(* IEC 61131-3 sources: MotionTestBenchMaster/Logical/00_AID/Libraries/Sidel_Libraries/Sidel (part 2) *)

(* ---- PID_FB.st ---- *)
FUNCTION_BLOCK PID_Cont
	VAR_RTInfo(enable:=TRUE);
	VAR_CycleCounter	:= MAX(1, VAR_CycleCounter + 1);

	TON_Cycle(	IN := TRUE,
				PT := IN_CycleTime - UDINT_TO_TIME(VAR_RTInfo.cycle_time / 1000));

	IF NOT TON_Cycle.Q THEN
		RETURN;
	END_IF

	VAR_CycleTime	:= (UDINT_TO_REAL(VAR_RTInfo.cycle_time) * VAR_CycleCounter) / 1000000.0;
	VAR_CycleCounter 	:= 0.0;
	memset(ADR(TON_Cycle), 0, SIZEOF(TON_Cycle));

	(*****************************************************************)
	(*************************SP MANAGE*******************************)
	(*****************************************************************)
	IF NOT VAR_FirstCycle THEN
		VAR_FirstCycle	:= TRUE;
		HMI.SPLocal		:= FALSE;
		OUT		:= 0.0;
		OUT_P	:= 0.0;
		OUT_I	:= 0.0;
		OUT_D	:= 0.0;
	END_IF

	IF EDGE(HMI.SPLocal) OR EDGEPOS(IN_Auto) THEN
		VAR_SlewInit	:= TRUE;
	END_IF

	IF VAR_SlewInit AND HMI.SPLocal THEN
		HMI.PV		:= IN_PV;
		LCRRamp.x	:= MIN(IN_PV, HMI.SP_Local);
		LCRRamp.set	:= TRUE;
	ELSIF VAR_SlewInit AND IN_Auto THEN
		HMI.PV		:= IN_PV;
		LCRRamp.x	:= MIN(IN_PV, IN_AutoSP);
		LCRRamp.set	:= TRUE;
	ELSIF HMI.SPLocal THEN
		HMI.PV		:= IN_PV;
		LCRRamp.x	:= HMI.SP_Local;
		LCRRamp.set	:= NOT HMI.ConfigSlewPresent;
	ELSIF IN_Auto THEN
		HMI.PV		:= IN_PV;
		LCRRamp.x	:= IN_AutoSP;
		LCRRamp.set := NOT HMI.ConfigSlewPresent;
	ELSE
		HMI.PV		:= 0.0;
		LCRRamp.x	:= 0.0;
		LCRRamp.set	:= TRUE;
	END_IF

	IF VAR_SlewInit AND LCRRamp.x_reached THEN
		VAR_SlewInit := FALSE;
	END_IF

	LCRRamp(
		enable	:= TRUE,
		dy_up	:= MAX(0.01, IN_SPSlew),
		dy_down := MAX(0.01, IN_SPSlew),
		y_min	:= 0.0,
		y_max	:= IN_MaxScale,
		y_set	:= LCRRamp.x
		);

	VAR_SPRamped := LCRRamp.y;

	(*****************************************************************)
	(***********************PID CONTROL*******************************)
	(*****************************************************************)
	IF IN_ConfigEngValue THEN
		LCRLimScal_PV(
			x	:= IN_PV,
			x1	:= 0.0,
			y1	:= 0.0,
			x2	:= IN_MaxScale,
			y2	:= 100.0
			);
		VAR_PV	:= LCRLimScal_PV.y;

		LCRLimScal_SP(
			x	:= VAR_SPRamped,
			x1	:= 0.0,
			y1	:= 0.0,
			x2	:= IN_MaxScale,
			y2	:= 100.0
			);
		VAR_SP	:= LCRLimScal_SP.y;
	ELSE
		VAR_SP	:= VAR_SPRamped;
		VAR_PV	:= IN_PV;
	END_IF

	IF IN_Reverse THEN
		OUT_Error := (VAR_PV - VAR_SP);
	ELSE
		OUT_Error := (VAR_SP - VAR_PV);
	END_IF

	(*****************************************************************)
	(********************PROPORTIONAL FACTOR**************************)
	(*****************************************************************)
	IF IN_Gain = 0 THEN
		VAR_GainError := OUT_Error;
	ELSE
		VAR_GainError := OUT_Error * IN_Gain;
	END_IF

	IF (IN_Auto OR HMI.SPLocal) THEN
		VAR_Proportional := VAR_GainError;
	ELSE
		VAR_Proportional := 0.0;
	END_IF

	OUT_P := VAR_Proportional;

	(*****************************************************************)
	(***********************INTEGRAL FACTOR***************************)
	(*****************************************************************)
	VAR_IntegralSaturation := (((OUT_P + OUT_I + OUT_D + IN_Disv) > IN_OutMax) AND OUT_Error > 0) OR (((OUT_P + OUT_I + OUT_D + IN_Disv) < IN_OutMin) AND OUT_Error < 0);
	VAR_IntegralBlock := IN_IntHold OR NOT (IN_Auto OR HMI.SPLocal) OR VAR_IntegralSaturation;  // integral block if saturated (anti wind up)

	VAR_Integral.IN_IntCycle := VAR_CycleTime;

	IF (IN_Auto OR HMI.SPLocal) AND IN_TI > 0 AND NOT IN_TIInit THEN
		IF EDGEPOS(IN_Auto OR HMI.SPLocal)THEN
			IF OUT > 0 THEN
				VAR_IntegralOut := OUT - OUT_P - IN_Disv;    (* Bumpless - Inizilize the Integral Component when the PID is setted in auto again *)
				VAR_Integral.IN_NewValue := VAR_IntegralOut;
				VAR_Integral(OUT_Integral := VAR_IntegralOut);
			END_IF
		ELSIF NOT VAR_IntegralBlock THEN
			VAR_Integral.IN_NewValue := VAR_GainError / IN_TI;
			//	VAR_IntegralOut := VAR_IntegralOut;
			IF VAR_Integral.IN_IntCycle > 0 THEN
				VAR_Integral(OUT_Integral := VAR_IntegralOut);
			END_IF
		END_IF
	ELSE
		IF IN_TIInit THEN
			VAR_IntegralOut := IN_TIInitValue;
		ELSE
			VAR_IntegralOut := 0.0;
		END_IF
	END_IF

	OUT_I := LIMIT((IN_OutMax * -1.0), VAR_IntegralOut, IN_OutMax);

	(*****************************************************************)
	(**********************DERIVATIVE FACTOR**************************)
	(*****************************************************************)
	IF (IN_Auto OR HMI.SPLocal) AND IN_TD >0 AND VAR_CycleTime > 0 THEN
		VAR_Derivative := ( VAR_GainError - VAR_OldError ) * IN_TD / VAR_CycleTime;
	ELSE
		VAR_Derivative := 0.0;
	END_IF
	VAR_OldError := VAR_GainError;

	OUT_D := VAR_Derivative;

	(*****************************************************************)
	(************************OUT CALCOLATION**************************)
	(*****************************************************************)
	IF HMI.Enable AND IN_ConfigPresent THEN
		OUT:= LIMIT(IN_OutMin, OUT_P + OUT_I + OUT_D + IN_Disv, IN_OutMax);
	ELSIF IN_FixOut THEN
		OUT:= LIMIT(IN_OutMin, IN_FixOutValue, IN_OutMax);
	ELSE
		OUT:= 0.0;
	END_IF

	(*****************************************************************)
	(*******************************HMI*******************************)
	(*****************************************************************)
	HMI.Enable			:= IN_Auto OR HMI.SPLocal;
	HMI.Mode			:= NOT HMI.SPLocal;
	HMI.SP_SlewRunning	:= LCRRamp.enable AND NOT LCRRamp.x_reached;

	HMI.ConfigPresent		:= IN_ConfigPresent;
	HMI.ConfigSlewPresent	:= IN_Slew;

	OUT_ActSP			:= VAR_SPRamped;
	HMI.SP_Actual		:= OUT_ActSP;
	HMI.SP_Target		:= IN_AutoSP;
	HMI.SP_Obtained		:= (IN_PV < (IN_AutoSP + IN_MaxDev)) AND (IN_PV > (IN_AutoSP - IN_MinDev));
	HMI.FF_OUT			:= IN_Disv;
	HMI.OUT				:= OUT;
END_FUNCTION_BLOCK

FUNCTION_BLOCK Integral
	OUT_Integral := OUT_Integral + ( VAR_OldValue + (IN_NewValue -  VAR_OldValue ) * 0.5 ) * IN_IntCycle;
	VAR_OldValue := IN_NewValue;
END_FUNCTION_BLOCK

(* ---- PID_FF_Mod.st ---- *)
FUNCTION_BLOCK PID_FF_Mod
	IF SP1_ON THEN
		FF_SP2_Save := IN_FF_SP2;
		IF FF_SP2_Save >= IN_FF_SP1 THEN
			FF_SP2_Save := IN_FF_SP1;
		END_IF
		FF_SP2_Time.PT := REAL_TO_TIME(IN_SP1_SP2_Time/1000);
	END_IF

	FF_SP2_Time.IN := SP1_ON;
	FF_SP2_Time();

	IF NOT IN_Reset AND IN_Enable THEN
		IF ( IN_Raise_Step_Counter >= IN_Raise_Step ) OR ( IN_Raise_Step_Counter >= 100 ) THEN
			Running := TRUE;
			Lower_Ramp := TRUE;
		END_IF
	END_IF

	IF (NOT IN_Enable AND (( IN_Lower_Step_Counter >= IN_Lower_Step ) OR ( IN_Lower_Step_Counter >= 100 )))
		OR IN_Reset THEN
		Running := FALSE;
		SP1_ON := FALSE;
		SP2_ON := FALSE;
	END_IF

	FF_SP1_Recipe := (IN_FF_SP1);
	FF_SP2_Recipe := (IN_FF_SP2);
	Speed := IN_Actual_Speed;
	Max_Speed := MAX(IN_Size_Speed, 1);

	FF_SP1_Val := FF_SP1_Recipe * Speed;
	FF_SP1_Val := FF_SP1_Val / Max_Speed;

	FF_SP2_Val := FF_SP2_Recipe * Speed;
	FF_SP2_Val := FF_SP2_Val / Max_Speed;

	IF NOT Running AND NOT Lower_Ramp THEN
		FF_value_Out := 0.0;
	ELSIF NOT Running THEN
		Ramp_Time := 200.0;
		Ramp_Speed_R := (IN_Ramp_Speed);
		Ramp_Value := Ramp_Value - ((Ramp_Time /1000.0) * Ramp_Speed_R );
		IF Ramp_Value <= 0 THEN
			Lower_Ramp := FALSE;
			Ramp_Value := 0;
		END_IF
		FF_value_Out := Ramp_Value;
	ELSIF SP2_ON THEN
		FF_value_Out := FF_SP2_Val;
		Ramp_Value := FF_SP2_Val;
	ELSIF FF_SP2_Time.Q THEN
		Ramp_Time := 200.0;
		Ramp_Speed_R := (IN_Ramp_Speed);
		Ramp_Value := Ramp_Value - ((Ramp_Time /1000.0) * Ramp_Speed_R );
		IF Ramp_Value <= FF_SP2_Val THEN
			SP2_ON := TRUE;
			Ramp_Value := FF_SP2_Val;
		END_IF
		FF_value_Out := Ramp_Value;
	ELSIF SP1_ON THEN
		FF_value_Out := FF_SP1_Val;
		Ramp_Value := FF_SP1_Val;
	ELSE
		Ramp_Time := 200.0;
		Ramp_Speed_R := (IN_Ramp_Speed);
		Ramp_Value := Ramp_Value + ((Ramp_Time /1000.0) * Ramp_Speed_R );
		FF_value_Out := Ramp_Value;
		IF Ramp_Value >= FF_SP1_Val THEN
			SP1_ON := TRUE;
		END_IF
	END_IF

	OUT_FF_Value := FF_value_Out;
	OUT_FF_Value_Int := REAL_TO_INT(FF_value_Out);
END_FUNCTION_BLOCK

(* ---- PID_FF_Pump.st ---- *)
FUNCTION_BLOCK PID_FF_Pump
//Pressure Head = (Frequency * Frequency * Kf ) - (Kpc * Flow * Flow)
//To find Kf:
//1. Container Block
//2. Filler Empty with Filling Valves Closed
//3. Search for right Kf until FF = PID Out

//To Find Kpc:
//1. Filler at Max Speed
//2. Filler full of containers, filling containers
//3. Search for right Kpc until FF = PID Out

//                   /^^^^^^^^^^^^^^^^^^^^^^^^^^^^^^^^^^^^^^^^^^^^
//Pump Frquency =  \/ ((Pressure Head) + Kpc * (Flow * Flow)) / Kf

//Pump Frequency [Hz]
//Pressure Head [mbar] --> mm
//Flow [m3/h]

IF NOT IN_Enable OR IN_Reset THEN
	OUT_FF	:= 0.0;
	RETURN;
END_IF

//Calculation of centrifugal force
//F_{cf}= m {\omega^2}{r} --> Omega is the Angular Velocity.
//Filler Angular Velocity
Omega := ((IN_Actual_Speed / IN_FV_Number) / (3600.0)) * 2.0 * 3.1415;

//Filler Radius
IF IN_Control_Type THEN //0=Control on Ring;1=Control on Product Pipe
	Radius := (IN_RingDiameter_mm / 2.0 / 1000.0);
ELSE
	Radius := 0.0;
END_IF

//Centrifugal Force [N], With Gravity Aceleration
IF IN_Control_Type THEN //0=Control on Ring;1=Control on Product Pipe
	CentrifugalForce := ((0.5 * Omega * Omega * Radius * Radius) / 9.81) * 1000.0;
ELSE
	CentrifugalForce := (((0.5 * Omega * Omega * Radius * Radius) / 9.81) * 1000.0)/100; //Convertion to mm of Product Pump In Ring Configuration
END_IF

IF IN_Control_Type THEN //0=Control on Ring;1=Control on Product Pipe
	Level_SP_Calculated := IN_Actual_SPmm + IN_PTF_FromFloor + IN_PTF_FromFV - CentrifugalForce;	//[mm] Of Water From The Floor To The SP Product Pump
ELSE
	Level_SP_Calculated := (IN_Actual_SPbar * 10197)- CentrifugalForce; // in test((IN_Actual_SPbar*1000) + IN_FV_FromFloor + 430 (*offset between fv and PTF on ring*)) - CentrifugalForce;	//[mm] Of Water From The Floor To The SP Product Pump In Ring Configuration
END_IF

IF IN_Control_Type THEN //0=Control on Ring;1=Control on Product Pipe
	PV_Product_Pump:= (IN_Actual_PVmm + IN_PTF_FromFloor + IN_PTF_FromFV) - IN_TankLevel_mm; //[mm] Of Water From The Floor on The PV Product Pump -Used For Pump Autotuning
ELSE
	PV_Product_Pump:= ((IN_Actual_PVbar * 1000)+ IN_FV_FromFloor + 430) - IN_TankLevel_mm; //[mm] Of Water From The Floor on The PV Product Pump In Ring Configuration
END_IF

//Hz For Actual Flowrate
Kpc_FlowRate_Filling := IN_Pump_Kpc * EXPT(((IN_FMCActualFlowrate/ 10.0) * 60.0) / 1000.0 , 2); //FF Calc on Filling Valves OPENED From FMC

//Real Set Point
Real_Level := Level_SP_Calculated - IN_TankLevel_mm;

//Calculated PV
IF IN_Control_Type THEN //0=Control on Ring;1=Control on Product Pipe
	Pid_PV_Calculated := (IN_Actual_PVmm + CentrifugalForce - IN_PTF_FromFV);
ELSE
	Pid_PV_Calculated := IN_Actual_PVbar;
END_IF

IF Pid_PV_Calculated > 0 THEN
	OUT_PID_PV := Pid_PV_Calculated;
ELSE
	OUT_PID_PV := 0.0;
END_IF

IF Pid_PV_Calculated > 0 THEN
	IF IN_Control_Type THEN //0=Control on Ring;1=Control on Product Pipe
		OUT_PID_SP := IN_Actual_SPmm + IN_PTF_FromFV - CentrifugalForce;
	ELSE
		OUT_PID_SP := IN_Actual_SPbar (*- (CentrifugalForce/1000)*);
	END_IF
ELSE
	OUT_PID_SP := 0.0;
END_IF

//Feed Forward Value for PID Control
IF SQRT((Kpc_FlowRate_Filling + Real_Level) / IN_Pump_Kf) >0 THEN
	OUT_FF := LIMIT(0,SQRT((Kpc_FlowRate_Filling + Real_Level) / IN_Pump_Kf),IN_Pump_OutMax);
ELSE
	OUT_FF := 0.0;
END_IF

//Detecting Wrong Setting
IF IN_Control_Type THEN //0=Control on Ring;1=Control on Product Pipe
	OUT_Error := IN_RingDiameter_mm =0.0 OR IN_PTF_FromFloor=0.0 OR IN_PTF_FromFV=0.0 OR IN_Pump_Kf=0.0 OR IN_Pump_Kpc=0.0 OR IN_Pump_OutMax=0.0;
ELSE
	OUT_Error := IN_FV_FromFloor=0.0 OR IN_Pump_Kf=0.0 OR IN_Pump_Kpc=0.0 OR IN_Pump_OutMax=0.0;
END_IF

END_FUNCTION_BLOCK

FUNCTION_BLOCK PID_FF_PumpH
//Pressure Head = (Frequency * Frequency * Kf ) - (Kpc * Flow * Flow)
//To find Kf:
//1. Container Block
//2. Filler Empty with Filling Valves Closed
//3. Search for right Kf until FF = PID Out

//To Find Kpc:
//1. Filler at Max Speed
//2. Filler full of containers, filling containers
//3. Search for right Kpc until FF = PID Out

//                  /^^^^^^^^^^^^^^^^^^^^^^^^^^^^^^^^^^^^^^^^^^^^
//Pump Frquency =  \/ ((Pressure Head) + Kpc * (Flow * Flow)) / Kf

//Pump Frequency [Hz]
//Pressure Head [mbar] --> mm
//Flow [m3/h]

IF NOT IN_Enable OR IN_Reset THEN
	OUT_FF	:= 0.0;
	RETURN;
END_IF

//Calculation of centrifugal force
//F_{cf}= m {\omega^2}{r} --> Omega is the Angular Velocity.
//Filler Angular Velocity
Omega := ((IN_Actual_Speed / IN_FV_Number) / (3600.0)) * 2.0 * 3.1415;

//Filler Radius
IF IN_Control_Type THEN //0=Control on Ring;1=Control on Product Pipe
	Radius := (IN_RingDiameter_mm / 2.0 / 1000.0);
ELSE
	Radius := 0.0;
END_IF

//Centrifugal Force [N], With Gravity Aceleration
IF IN_Control_Type THEN //0=Control on Ring;1=Control on Product Pipe
	CentrifugalForce := ((0.5 * Omega * Omega * Radius * Radius) / 9.81) * 1000.0;
ELSE
	CentrifugalForce := (((0.5 * Omega * Omega * Radius * Radius) / 9.81) * 1000.0)/100; //Convertion to mm of Product Pump In Ring Configuration
END_IF

//MAX Filling Time
MAX_FillingTime := (1000.0 / (IN_Recipe_Speed /3600.0)) * IN_FMCStepExitCam;

//Actual Filling Time
IF IN_FMCAverFillingTime >= 0 THEN
	Calculated_FillingTime := IN_FMCAverFillingTime;
ELSE
	Calculated_FillingTime := IN_PumpMaxFillingTime;
END_IF

FillingTime := MIN(Calculated_FillingTime,MAX_FillingTime);

//MAX Containers Number Into Filling Zone (Used only to control the value from the FMC "ITC_FMC_Tot_FV_Actual_In_Filling")
MAX_ContainersNumber := ((IN_Recipe_Speed * FillingTime / 3600000.0) - IN_FMCStepStartFilling);

IF IN_Control_Type THEN //0=Control on Ring;1=Control on Product Pipe
	Level_SP_Calculated := IN_Actual_SPmm + IN_PTF_FromFloor + IN_PTF_FromFV - CentrifugalForce;	//[mm] Of Water From The Floor To The SP Product Pump
ELSE
	Level_SP_Calculated := ((IN_Actual_SPbar*1000)+ IN_FV_FromFloor + 430(*offset between fv and PTF on ring*)) - CentrifugalForce;	//[mm] Of Water From The Floor To The SP Product Pump In Ring Configuration
END_IF

IF IN_Control_Type THEN //0=Control on Ring;1=Control on Product Pipe
	PV_Product_Pump:= (IN_Actual_PVmm + IN_PTF_FromFloor + IN_PTF_FromFV) - IN_TankLevel_mm; //[mm] Of Water From The Floor on The PV Product Pump -Used For Pump Autotuning
ELSE
	PV_Product_Pump:= ((IN_Actual_PVbar *1000)+ IN_FV_FromFloor + 430) - IN_TankLevel_mm; //[mm] Of Water From The Floor on The PV Product Pump In Ring Configuration
END_IF

//Hz For Actual Flowrate
Kpc_FlowRate_Filling := IN_Pump_Kpc * EXPT(((IN_FMCActualFlowrate/ 10.0) * 60.0) / 1000.0 , 2); //FF Calc on Filling Valves OPENED From FMC

//Real Set Point
Real_Level := Level_SP_Calculated - IN_TankLevel_mm;

//Centrifugal Force
OUT_Centifrugal := CentrifugalForce;

//Feed Forward Value for PID Control
IF SQRT((Kpc_FlowRate_Filling + Real_Level) / IN_Pump_Kf) >0 THEN
	OUT_FF := LIMIT(0,SQRT((Kpc_FlowRate_Filling + Real_Level) / IN_Pump_Kf),IN_Pump_OutMax);
ELSE
	OUT_FF := 0.0;
END_IF

//Detecting Wrong Setting
IF IN_Control_Type THEN //0=Control on Ring;1=Control on Product Pipe
OUT_Error := IN_RingDiameter_mm =0.0 OR IN_PTF_FromFloor=0.0 OR IN_PTF_FromFV=0.0 OR
			 IN_Pump_Kf=0.0 OR IN_Pump_Kpc=0.0 OR IN_Pump_OutMax=0.0 OR IN_FMCAverFillingTime=0.0 OR
			 IN_FMCStepStartFilling= 0.0 OR IN_FMCStepExitCam=0.0;
ELSE
	OUT_Error := IN_FV_FromFloor=0.0 OR IN_Pump_Kf=0.0 OR IN_Pump_Kpc=0.0 OR IN_Pump_OutMax=0.0;
END_IF

END_FUNCTION_BLOCK

(* ---- RCP_Management.st ---- *)
FUNCTION_BLOCK RCP_Management
	IF NOT VAR_FirstCycle THEN
		IF (memcmp(IN_AdrPLCRecipe, IN_AdrHMIRecipe, IN_SizePLCRecipe) <> 0) OR (memcmp(IN_AdrHMIRecipe, IN_AdrPLCRecipe, IN_SizeHMIRecipe) <> 0) THEN
			OUT_ParameterError := TRUE;
			RETURN;
		ELSE
			VAR_FirstCycle := TRUE;
		END_IF
	END_IF

	TMR_tonRCP_WaitStart.IN			:= FALSE;
	TMR_tonRCP_DownloadTimeOut.IN	:= FALSE;

	CASE OUT_Step OF

		Wait_Download:
			RCP_Manag.RequestedRecipeName	:= IN_RequestedRCP;
			TMR_tonRCP_WaitStart.IN			:= IN_DownloadRequest OR RCP_Manag.Started;
			TMR_tonRCP_WaitStart.PT			:= t#500ms;

			IF TMR_tonRCP_WaitStart.Q THEN
				OUT_Step := Download_Request;
			END_IF

			IF RCP_Manag.EditOnlineActive THEN
				OUT_Step := Edit_Online;
			END_IF

		Download_Request:
			RCP_Manag.RequestedRecipeName 	:= IN_RequestedRCP;
			RCP_Manag.DownloadRequest		:= IN_DownloadRequest;

			IF (RCP_Manag.Started AND RCP_Manag.Ended) THEN
				OUT_Step := Copy_To_Internal;
			END_IF

			TMR_tonRCP_DownloadTimeOut.IN	:= NOT RCP_Manag.Ended OR (NOT RCP_Manag.Started AND RCP_Manag.Ended);
			TMR_tonRCP_DownloadTimeOut.PT	:= t#10s;

			IF TMR_tonRCP_DownloadTimeOut.Q THEN
				OUT_Step := Download_Error;
			END_IF

		Copy_To_Internal:
			RCP_Manag.DownloadRequest := FALSE;

			IF (memcmp(IN_AdrPLCRecipe,IN_AdrHMIRecipe,IN_SizePLCRecipe) <> 0) THEN
				memcpy(IN_AdrPLCRecipe,IN_AdrHMIRecipe,IN_SizePLCRecipe);
			END_IF

			IF IN_DownloadRequest THEN
				IF (IN_RequestedRCP = RCP_Manag.ActiveRecipeName) THEN	// Check Request Recipe Name
					IF (memcmp(IN_AdrPLCRecipe,IN_AdrHMIRecipe,IN_SizePLCRecipe) = 0) THEN
						OUT_Step := Download_Done;
					END_IF
				END_IF
			ELSE
				OUT_Step := Download_Done;
			END_IF

			TMR_tonRCP_DownloadTimeOut.IN := (IN_RequestedRCP <> RCP_Manag.ActiveRecipeName);
			TMR_tonRCP_DownloadTimeOut.PT := t#5s;

			IF TMR_tonRCP_DownloadTimeOut.Q THEN
				OUT_Step := Download_Error;
			END_IF

		Download_Done:
			RCP_Manag.Received	:= TRUE;
			OUT_RecipeLoaded	:= TRUE;

			IF (NOT RCP_Manag.Ended AND NOT (IN_DownloadRequest OR RCP_Manag.Started)) THEN
				OUT_Step := Clear_Cmd;
			END_IF

		Clear_Cmd:
			RCP_Manag.Received := FALSE;
			RCP_Manag.RequestedRecipeName := '';
			OUT_Step := Wait_Download;

		Edit_Online:
			IF RCP_Manag.EditOnlineActive THEN
				IF (memcmp(IN_AdrPLCRecipe,IN_AdrHMIRecipe,IN_SizePLCRecipe) <> 0) THEN
					memcpy(IN_AdrPLCRecipe,IN_AdrHMIRecipe,IN_SizePLCRecipe);
				END_IF
			ELSE
				OUT_Step := Clear_Cmd;
			END_IF

		Download_Error:
			RCP_Manag.Received := FALSE;
			RCP_Manag.DownloadRequest := FALSE;
			RCP_Manag.Started := FALSE;
			RCP_Manag.Ended := FALSE;
			RCP_Manag.RequestedRecipeName := '';

			TMR_tonRCP_WaitRestart.IN := IN_DownloadRequest OR RCP_Manag.Started;
			TMR_tonRCP_WaitRestart.PT := t#3s;

			IF TMR_tonRCP_WaitRestart.Q THEN
				OUT_Step := Download_Request;
			END_IF

			IF NOT IN_DownloadRequest AND NOT RCP_Manag.Started THEN
				OUT_Step := Wait_Download;
			END_IF
	END_CASE

	IF OUT_Step <> VAR_Step_old THEN
		TMR_tonRCP_WaitStart.IN			:= FALSE;
		TMR_tonRCP_DownloadTimeOut.IN	:= FALSE;
		VAR_Step_old := OUT_Step;
	END_IF

	TMR_tonRCP_WaitStart();
	TMR_tonRCP_DownloadTimeOut();
END_FUNCTION_BLOCK

(* ---- Sequencer.st ---- *)
FUNCTION_BLOCK Sequencer_v1
	VAR_ChangeInProgress := OUT_JMP_Step <> IN_Step;

	IF VAR_ChangeInProgress THEN
		memset(ADR(TON_Time),	0,	SIZEOF(TON_Time));
		memset(ADR(T_Time),		0,	SIZEOF(T_Time));
		memset(ADR(TO_Time),	0,	SIZEOF(TO_Time));
		OUT_JMP_StepPrevious := OUT_JMP_Step ;
	END_IF

	//Volatile Timer
	TON_Time(
	IN := IN_StepConfig.TON_TimeSTART AND NOT VAR_ChangeInProgress AND NOT IN_Pause_Request,
	PT := UINT_TO_TIME(IN_StepConfig.TON_TimePr * 1000)
	);
	OUT_TON_Time_END := TON_Time.Q;

	//Retentive Counter
	T_Time(
	CU 		:= IN_T_TimeClock AND IN_StepConfig.T_TimeSTART AND NOT IN_StepConfig.T_TimeSTOP AND NOT IN_Pause_Request,
	RESET 	:= IN_StepConfig.T_TimeRESET OR VAR_ChangeInProgress,
	PV 		:= IN_StepConfig.T_TimePr
	);
	OUT_T_Time_END := T_Time.Q;

	//Volatile Timeout
	TO_Time(
	IN := NOT VAR_ChangeInProgress,
	PT := UINT_TO_TIME(IN_StepConfig.TO_TimePr * 1000)
	);
	OUT_TO_Time_END := TO_Time.Q;

	//Reset counter Initialized to wait counter reset from Filler
	IF VAR_ChangeInProgress THEN
		VAR_CounterInitialized := FALSE;
	END_IF

	//Eneble Laps Counter Request only if the counter is initialized
	IF NOT VAR_CounterInitialized THEN
		OUT_LapsCounterRequest := FALSE;
	ELSIF IN_StepConfig.Laps_Counter_Enable THEN
		OUT_LapsCounterRequest := TRUE;
	END_IF

	//Step Counter is initialized when the value is 0
	IF IN_StepCounter = 0 THEN
		VAR_CounterInitialized := TRUE;
	END_IF

	//Laps Progress
	OUT_Laps_Progress := (IN_StepCounter / MAX(1, IN_FillingValveNr));

	//Laps Expired
	OUT_Laps_Done := OUT_Laps_Progress >= IN_StepConfig.Laps_Request AND IN_StepCounter > 0 AND IN_StepConfig.Laps_Counter_Enable;

	OUT_JMP_Step 	:= IN_Step;
	OUT_HMI_ID		:= IN_StepConfig.HMI_ID;

	//Cycles
	IF CyclesCounter >= IN_StepConfig.Cycle_Pr THEN
		OUT_Cycles_Done := TRUE;
	ELSE
		OUT_Cycles_Done:= FALSE;
	END_IF

	//Timers Visualization
	OUT_StepTimePr_TON  := REAL_TO_UINT(TIME_TO_REAL(TON_Time.PT) / 1000.0);
	OUT_StepTimePr_T    := T_Time.PV;
	OUT_StepTimeCV_TON	:= REAL_TO_UINT(TIME_TO_REAL(TON_Time.ET) / 1000.0);
	OUT_StepTimeCV_T    := T_Time.CV;

END_FUNCTION_BLOCK

FUNCTION_BLOCK Sequencer_v2
	VAR_ChangeInProgress := OUT_StepActual <> IN_Step; //v2

	IF VAR_ChangeInProgress THEN
		memset(ADR(TON_Time),	0,	SIZEOF(TON_Time));
		memset(ADR(T_Time),		0,	SIZEOF(T_Time));
		memset(ADR(TO_Time),	0,	SIZEOF(TO_Time));
		OUT_StepPrevious := OUT_StepActual; //v2
	END_IF

	//Volatile Timer
	TON_Time(
	IN := IN_StepConfig.TON_TimeSTART AND NOT VAR_ChangeInProgress AND NOT IN_Pause_Request,
	PT := UINT_TO_TIME(IN_StepConfig.TON_TimePr * 1000)
	);
	OUT_TON_Time_END := TON_Time.Q;

	//Retentive Counter
	T_Time(
	CU 		:= IN_T_TimeClock AND IN_StepConfig.T_TimeSTART AND NOT IN_StepConfig.T_TimeSTOP AND NOT IN_Pause_Request,
	RESET 	:= IN_StepConfig.T_TimeRESET OR VAR_ChangeInProgress,
	PV 		:= IN_StepConfig.T_TimePr
	);
	OUT_T_Time_END := T_Time.Q;

	//Volatile Timeout
	TO_Time(
	IN := NOT VAR_ChangeInProgress,
	PT := UINT_TO_TIME(IN_StepConfig.TO_TimePr * 1000)
	);
	OUT_TO_Time_END := TO_Time.Q;

	//Progressive Time v2
	T_StepProgressiveTime(
	IN := NOT VAR_ChangeInProgress,
	PT := T#24d,
	);

	//Reset counter Initialized to wait counter reset from Filler
	IF VAR_ChangeInProgress THEN
		VAR_CounterInitialized := FALSE;
	END_IF

	//Eneble Laps Counter Request only if the counter is initialized
	IF NOT VAR_CounterInitialized THEN
		OUT_LapsCounterRequest := FALSE;
	ELSIF IN_StepConfig.Laps_Counter_Enable THEN
		OUT_LapsCounterRequest := TRUE;
	END_IF

	//Step Counter is initialized when the value is 0
	IF IN_StepCounter = 0 THEN
		VAR_CounterInitialized := TRUE;
	END_IF

	//Laps Progress
	OUT_Laps_Progress := (IN_StepCounter / MAX(1, IN_FillingValveNr));

	//Laps Expired
	OUT_Laps_Done := OUT_Laps_Progress >= IN_StepConfig.Laps_Request AND IN_StepCounter > 0 AND IN_StepConfig.Laps_Counter_Enable;

	OUT_StepActual 	:= IN_Step; //v2
	OUT_HMI_ID		:= IN_StepConfig.HMI_ID;

	//Cycles
	IF CyclesCounter >= IN_StepConfig.Cycle_Pr THEN
		OUT_Cycles_Done := TRUE;
	ELSE
		OUT_Cycles_Done:= FALSE;
	END_IF

	//Timers Visualization
	OUT_StepTimePr_TON  	:= REAL_TO_UINT(TIME_TO_REAL(TON_Time.PT) / 1000.0);
	OUT_StepTimePr_T    	:= T_Time.PV;
	OUT_StepTimeCV_TON		:= REAL_TO_UINT(TIME_TO_REAL(TON_Time.ET) / 1000.0);
	OUT_StepTimeCV_T    	:= T_Time.CV;
	OUT_StepProgressiveTime	:= REAL_TO_UINT(TIME_TO_REAL(T_StepProgressiveTime.ET) / 1000.0); //v2

END_FUNCTION_BLOCK

(* ---- Sidel.fun ---- *)
FUNCTION FC_Parity : BOOL (*TRUE = Even - FALSE = ODD*)
	VAR_INPUT
		IN_Value : DINT;
	END_VAR
END_FUNCTION

FUNCTION_BLOCK AlarmScheduler (*V4.A.A.1.6.13*)
	VAR_INPUT
		AlarmAreaCfg : ARRAY[0..24] OF AlarmAreaCfg_Type;
		AdrAlarm : UDINT;
		AdrAlarmCFG : UDINT;
		AdrAlarmOldStatus : UDINT;
		AdrHMI : UDINT;
	END_VAR
	VAR_OUTPUT
		AlarmAction : ActionSum_Type;
	END_VAR
	VAR_IN_OUT
		FirstAlarmActive : AlarmCFG_Type;
		FirstExternalAlarmActive : AlarmCFG_Type;
		FirstCriticalAlarmActive : AlarmCFG_Type; (*V4.A.A.1.7.0*)
		FirstAlertAlarmActive : AlarmCFG_Type; (*V4.A.A.1.7.0*)
		FirstExtCriticalAlarmActive : AlarmCFG_Type; (*V4.A.A.1.7.0*)
		FirstExtAlertAlarmActive : AlarmCFG_Type; (*V4.A.A.1.7.0*)
		FirstCsAlarmActive : AlarmCFG_Type; (*V4.A.A.1.7.0*)
		CriticalAcknoledgeRequest : BOOL;
		AlarmAcknoledgeRequest : BOOL;
	END_VAR
	VAR
		Alarm : REFERENCE TO AlarmCmd_Type;
		AlarmOldStatus : REFERENCE TO BOOL;
		AlarmCFG : REFERENCE TO AlarmCFG_Type;
		HMI : REFERENCE TO BYTE;
		AlarmActionTemp : ActionSum_Type;
		i : UINT;
		x : UINT;
	END_VAR
END_FUNCTION_BLOCK

FUNCTION_BLOCK FirstAlarmCombiner (*V4.A.A.1.6.13*)
	VAR_INPUT
		SkidAlarmFrom : UINT := 1;
		SkidAlarmTo : UINT;
		SkidFirstAlarm : INT;
		SkidFirstExternalAlarm : INT;
	END_VAR
	VAR_IN_OUT
		FirstAlarmActive : AlarmCFG_Type;
		FirstExternalAlarmActive : AlarmCFG_Type;
	END_VAR
END_FUNCTION_BLOCK

FUNCTION_BLOCK AnalogTotalizer
	VAR_INPUT
		IN_Pulse : BOOL;
		IN_AnalogPV : REAL;
		IN_PulseWeight : REAL;
		IN_ConfigType : USINT; (*Configuaration Time to mapping if analog value is used
(0 = Pulse, 1 = Hours, 2 = Minutes, 3 = Seconds)*)
		IN_Reset : BOOL; (*Reset totalizer*)
	END_VAR
	VAR_IN_OUT
		OUT_TotalCounter : REAL; (*Out Total Counter*)
	END_VAR
	VAR
		RTInfo : RTInfo;
		VAR_AuxPulse : REAL;
		zzEdge00000 : BOOL;
	END_VAR
END_FUNCTION_BLOCK

FUNCTION_BLOCK CyclicActivation
	VAR_INPUT
		IN_CycleTime : TIME;
	END_VAR
	VAR_OUTPUT
		OUT_A : BOOL;
		OUT_B : BOOL;
	END_VAR
	VAR
		TMR_TON_CycleA : TON;
		TMR_TON_CycleB : TON;
		VAR_RtInfo : RTInfo;
		VAR_CycleCounter : REAL;
		VAR_CycleTime : REAL;
		VAR_Cycle : BOOL;
	END_VAR
END_FUNCTION_BLOCK

FUNCTION ComboBoxString : BOOL
	VAR_INPUT
		IN_ElementsStructure : ARRAY[0..16] OF HMI_ComboBoxElements_Type;
		OUT_ComboString : REFERENCE TO STRING[500];
	END_VAR
	VAR
		VAR_ElementsIndex : USINT;
		VAR_StrIndex : STRING[2];
		VAR_StrComma : STRING[1];
		VAR_StrSemicolun : STRING[1];
	END_VAR
END_FUNCTION

FUNCTION LftConAirPressSp : REAL
	VAR_INPUT
		RcpPressureSp : REAL;
		RcpCanDiameter : REAL;
	END_VAR
	VAR CONSTANT
		CST_PistonDiameterExt : REAL := 40.0; (*[mm]*)
		CST_PistonDiameterInt : REAL := 16.0; (*[mm]*)
		CST_PistonSpringStrengthRse : REAL := 120.0; (*[N]*)
	END_VAR
	VAR
		VAR_PistonSurface : REAL; (*[mm2]*)
		VAR_DeltaPProduct : REAL; (*[N]*)
		VAR_DeltaPrexPist : REAL; (*[bar]*)
		VAR_PbasePiston : REAL; (*[bar]*)
	END_VAR
END_FUNCTION

FUNCTION_BLOCK FB_Blinker
	VAR_INPUT
		IN_Freq : REAL;
	END_VAR
	VAR_OUTPUT
		OUT : BOOL;
	END_VAR
	VAR
		TMR_TON_OnDelay : TON;
		TMR_TON_OffDelay : TON;
		VAR_TimeValue : TIME;
	END_VAR
END_FUNCTION_BLOCK

FUNCTION_BLOCK FB_HMI_ITC_Start
	VAR_IN_OUT
		HMI_Data : HMI_ITC_Data_Type;
		AnalogIndexIn : UINT;
		DigitalIndexIn : UINT;
		AnalogIndexOut : UINT;
		DigitalIndexOut : UINT;
	END_VAR
	VAR
		i : UINT;
	END_VAR
END_FUNCTION_BLOCK

FUNCTION_BLOCK FB_HMI_ITC_DigitalBool
	VAR_INPUT
		IN_Visibility : BOOL;
		IN_ReadOnly : BOOL;
		IN_Wait : BOOL;
		IN_Alarm : BOOL;
		IN_IOType : BOOL; (*0: INPUT 1: OUTPUT*)
		IN_Description : STRING[100];
		IN_HMIAutoForce : BOOL;
	END_VAR
	VAR_OUTPUT
		OUT_Man : BOOL;
		OUT_ManValue : BOOL;
	END_VAR
	VAR_IN_OUT
		ITC_IO : BOOL;
		ITC : BOOL;
		HMI_Data : HMI_ITC_Data_Type;
		HMI_Page : HMI_ITC_Page_Type;
		Index : UINT;
	END_VAR
	VAR
		VAR_Auto : BOOL := TRUE;
		VAR_Man : BOOL := FALSE;
		VAR_PageSwitch : BOOL := TRUE;
		VAR_ProgressiveId : UINT;
		VAR_OldPage : USINT;
		zzEdge00000 : BOOL;
		zzEdge00001 : BOOL;
		zzEdge00002 : BOOL;
		zzEdge00003 : BOOL;
	END_VAR
END_FUNCTION_BLOCK

FUNCTION_BLOCK FB_HMI_ITC_DigitalByte
	VAR_INPUT
		IN_Visibility : BOOL;
		IN_ReadOnly : BOOL;
		IN_Wait : BOOL;
		IN_Alarm : BOOL;
		IN_IOType : BOOL; (*0: INPUT 1: OUTPUT*)
		IN_Description : STRING[100];
		IN_HMIAutoForce : BOOL;
		IN_BitNumber : INT;
	END_VAR
	VAR_OUTPUT
		OUT_Man : BOOL;
		OUT_ManValue : BOOL;
	END_VAR
	VAR_IN_OUT
		ITC_IO : BYTE;
		ITC : BOOL;
		HMI_Data : HMI_ITC_Data_Type;
		HMI_Page : HMI_ITC_Page_Type;
		Index : UINT;
	END_VAR
	VAR
		VAR_Auto : BOOL := TRUE;
		VAR_Man : BOOL := FALSE;
		VAR_PageSwitch : BOOL := TRUE;
		VAR_ProgressiveId : UINT;
		VAR_BitArray : ARRAY[0..7] OF BOOL;
		VAR_BitIndex : USINT;
		VAR_OldPage : USINT;
		zzEdge00000 : BOOL;
		zzEdge00001 : BOOL;
		zzEdge00002 : BOOL;
		zzEdge00003 : BOOL;
	END_VAR
END_FUNCTION_BLOCK

FUNCTION_BLOCK FB_HMI_ITC_DigitalUsint
	VAR_INPUT
		IN_Visibility : BOOL;
		IN_ReadOnly : BOOL;
		IN_Wait : BOOL;
		IN_Alarm : BOOL;
		IN_IOType : BOOL; (*0: INPUT 1: OUTPUT*)
		IN_Description : STRING[100];
		IN_HMIAutoForce : BOOL;
		IN_BitNumber : INT;
	END_VAR
	VAR_OUTPUT
		OUT_Man : BOOL;
		OUT_ManValue : BOOL;
	END_VAR
	VAR_IN_OUT
		ITC_IO : USINT;
		ITC : BOOL;
		HMI_Data : HMI_ITC_Data_Type;
		HMI_Page : HMI_ITC_Page_Type;
		Index : UINT;
	END_VAR
	VAR
		VAR_Auto : BOOL := TRUE;
		VAR_Man : BOOL := FALSE;
		VAR_PageSwitch : BOOL := TRUE;
		VAR_ProgressiveId : UINT;
		VAR_BitArray : ARRAY[0..7] OF BOOL;
		VAR_BitIndex : USINT;
		VAR_OldPage : USINT;
		zzEdge00000 : BOOL;
		zzEdge00001 : BOOL;
		zzEdge00002 : BOOL;
		zzEdge00003 : BOOL;
	END_VAR
END_FUNCTION_BLOCK

FUNCTION_BLOCK FB_HMI_ITC_DigitalInt
	VAR_INPUT
		IN_Visibility : BOOL;
		IN_ReadOnly : BOOL;
		IN_Wait : BOOL;
		IN_Alarm : BOOL;
		IN_IOType : BOOL; (*0: INPUT 1: OUTPUT*)
		IN_Description : STRING[100];
		IN_HMIAutoForce : BOOL;
		IN_BitNumber : INT;
	END_VAR
	VAR_OUTPUT
		OUT_Man : BOOL;
		OUT_ManValue : BOOL;
	END_VAR
	VAR_IN_OUT
		ITC_IO : INT;
		ITC : BOOL;
		HMI_Data : HMI_ITC_Data_Type;
		HMI_Page : HMI_ITC_Page_Type;
		Index : UINT;
	END_VAR
	VAR
		VAR_Auto : BOOL := TRUE;
		VAR_Man : BOOL := FALSE;
		VAR_PageSwitch : BOOL := TRUE;
		VAR_ProgressiveId : UINT;
		VAR_BitArray : ARRAY[0..15] OF BOOL;
		VAR_BitIndex : USINT;
		VAR_OldPage : USINT;
		zzEdge00000 : BOOL;
		zzEdge00001 : BOOL;
		zzEdge00002 : BOOL;
		zzEdge00003 : BOOL;
	END_VAR
END_FUNCTION_BLOCK

FUNCTION_BLOCK FB_HMI_ITC_AnalogByte
	VAR_INPUT
		IN_Visibility : BOOL;
		IN_ReadOnly : BOOL;
		IN_Wait : BOOL;
		IN_IOType : BOOL; (*0: INPUT 1: OUTPUT*)
		IN_Description : STRING[100];
		IN_MinValue : REAL;
		IN_MaxValue : REAL;
		IN_Unit : STRING[10];
		IN_HMIAutoForce : BOOL;
	END_VAR
	VAR_OUTPUT
		OUT_Man : BOOL;
		OUT_ManValue : BYTE;
	END_VAR
	VAR_IN_OUT
		ITC_IO : BYTE;
		ITC : BYTE;
		HMI_Data : HMI_ITC_Data_Type;
		HMI_Page : HMI_ITC_Page_Type;
		Index : UINT;
	END_VAR
	VAR
		VAR_Man : BOOL := FALSE;
		VAR_ManValue : BYTE := 0;
		VAR_PageSwitch : BOOL := TRUE;
		VAR_ProgressiveId : UINT;
		VAR_OldPage : USINT;
	END_VAR
END_FUNCTION_BLOCK

FUNCTION_BLOCK FB_HMI_ITC_AnalogUsint
	VAR_INPUT
		IN_Visibility : BOOL;
		IN_ReadOnly : BOOL;
		IN_Wait : BOOL;
		IN_IOType : BOOL; (*0: INPUT 1: OUTPUT*)
		IN_Description : STRING[100];
		IN_MinValue : REAL;
		IN_MaxValue : REAL;
		IN_Unit : STRING[10];
		IN_HMIAutoForce : BOOL;
	END_VAR
	VAR_OUTPUT
		OUT_Man : BOOL;
		OUT_ManValue : USINT;
	END_VAR
	VAR_IN_OUT
		ITC_IO : USINT;
		ITC : USINT;
		HMI_Data : HMI_ITC_Data_Type;
		HMI_Page : HMI_ITC_Page_Type;
		Index : UINT;
	END_VAR
	VAR
		VAR_Man : BOOL := FALSE;
		VAR_ManValue : USINT := 0;
		VAR_PageSwitch : BOOL := TRUE;
		VAR_ProgressiveId : UINT;
		VAR_OldPage : USINT;
	END_VAR
END_FUNCTION_BLOCK

FUNCTION_BLOCK FB_HMI_ITC_AnalogInt
	VAR_INPUT
		IN_Visibility : BOOL;
		IN_ReadOnly : BOOL;
		IN_Wait : BOOL;
		IN_IOType : BOOL; (*0: INPUT 1: OUTPUT*)
		IN_Description : STRING[100];
		IN_MinValue : REAL;
		IN_MaxValue : REAL;
		IN_Unit : STRING[10];
		IN_HMIAutoForce : BOOL;
	END_VAR
	VAR_OUTPUT
		OUT_Man : BOOL;
		OUT_ManValue : INT;
	END_VAR
	VAR_IN_OUT
		ITC_IO : INT;
		ITC : INT;
		HMI_Data : HMI_ITC_Data_Type;
		HMI_Page : HMI_ITC_Page_Type;
		Index : UINT;
	END_VAR
	VAR
		VAR_Man : BOOL := FALSE;
		VAR_Value : INT;
		VAR_ManValue : INT := 0;
		VAR_PageSwitch : BOOL := TRUE;
		VAR_ProgressiveId : UINT;
		VAR_OldPage : USINT;
	END_VAR
END_FUNCTION_BLOCK

FUNCTION_BLOCK FB_HMI_ITC_AnalogIntOverUsint
	VAR_INPUT
		IN_Visibility : BOOL;
		IN_ReadOnly : BOOL;
		IN_Wait : BOOL;
		IN_IOType : BOOL; (*0: INPUT 1: OUTPUT*)
		IN_Description : STRING[100];
		IN_MinValue : REAL;
		IN_MaxValue : REAL;
		IN_Unit : STRING[10];
		IN_HMIAutoForce : BOOL;
	END_VAR
	VAR_OUTPUT
		OUT_Man : BOOL;
		OUT_ManValue : INT;
	END_VAR
	VAR_IN_OUT
		ITC_IO : USINT;
		ITC : INT;
		HMI_Data : HMI_ITC_Data_Type;
		HMI_Page : HMI_ITC_Page_Type;
		Index : UINT;
	END_VAR
	VAR
		VAR_Man : BOOL := FALSE;
		VAR_RawValue : INT;
		VAR_Value : INT;
		VAR_ManValue : INT := 0;
		VAR_PageSwitch : BOOL := TRUE;
		VAR_ProgressiveId : UINT;
		VAR_OldPage : USINT;
	END_VAR
END_FUNCTION_BLOCK

FUNCTION_BLOCK FB_HMI_ITC_AnalogUintOverUsint
	VAR_INPUT
		IN_Visibility : BOOL;
		IN_ReadOnly : BOOL;
		IN_Wait : BOOL;
		IN_IOType : BOOL; (*0: INPUT 1: OUTPUT*)
		IN_Description : STRING[100];
		IN_MinValue : REAL;
		IN_MaxValue : REAL;
		IN_Unit : STRING[10];
		IN_HMIAutoForce : BOOL;
	END_VAR
	VAR_OUTPUT
		OUT_Man : BOOL;
		OUT_ManValue : UINT;
	END_VAR
	VAR_IN_OUT
		ITC_IO : USINT;
		ITC : UINT;
		HMI_Data : HMI_ITC_Data_Type;
		HMI_Page : HMI_ITC_Page_Type;
		Index : UINT;
	END_VAR
	VAR
		VAR_Man : BOOL := FALSE;
		VAR_RawValue : UINT;
		VAR_Value : UINT;
		VAR_ManValue : UINT := 0;
		VAR_PageSwitch : BOOL := TRUE;
		VAR_ProgressiveId : UINT;
		VAR_OldPage : USINT;
	END_VAR
END_FUNCTION_BLOCK

FUNCTION_BLOCK FB_HMI_ITC_AnalogDInt
	VAR_INPUT
		IN_Visibility : BOOL;
		IN_ReadOnly : BOOL;
		IN_Wait : BOOL;
		IN_IOType : BOOL; (*0: INPUT 1: OUTPUT*)
		IN_Description : STRING[100];
		IN_MinValue : REAL;
		IN_MaxValue : REAL;
		IN_Unit : STRING[10];
		IN_HMIAutoForce : BOOL;
	END_VAR
	VAR_OUTPUT
		OUT_Man : BOOL;
		OUT_ManValue : DINT;
	END_VAR
	VAR_IN_OUT
		ITC_IO : DINT;
		ITC : DINT;
		HMI_Data : HMI_ITC_Data_Type;
		HMI_Page : HMI_ITC_Page_Type;
		Index : UINT;
	END_VAR
	VAR
		VAR_Man : BOOL := FALSE;
		VAR_Value : DINT;
		VAR_ManValue : DINT := 0;
		VAR_PageSwitch : BOOL := TRUE;
		VAR_ProgressiveId : UINT;
		VAR_OldPage : USINT;
	END_VAR
END_FUNCTION_BLOCK

FUNCTION_BLOCK FB_HMI_ITC_AnalogUdint
	VAR_INPUT
		IN_Visibility : BOOL;
		IN_ReadOnly : BOOL;
		IN_Wait : BOOL;
		IN_IOType : BOOL; (*0: INPUT 1: OUTPUT*)
		IN_Description : STRING[100];
		IN_MinValue : REAL;
		IN_MaxValue : REAL;
		IN_Unit : STRING[10];
		IN_HMIAutoForce : BOOL;
	END_VAR
	VAR_OUTPUT
		OUT_Man : BOOL;
		OUT_ManValue : UDINT;
	END_VAR
	VAR_IN_OUT
		ITC_IO : UDINT;
		ITC : UDINT;
		HMI_Data : HMI_ITC_Data_Type;
		HMI_Page : HMI_ITC_Page_Type;
		Index : UINT;
	END_VAR
	VAR
		VAR_Man : BOOL := FALSE;
		VAR_Value : UDINT;
		VAR_ManValue : UDINT := 0;
		VAR_PageSwitch : BOOL := TRUE;
		VAR_ProgressiveId : UINT;
		VAR_OldPage : USINT;
	END_VAR
END_FUNCTION_BLOCK

FUNCTION_BLOCK FB_HMI_ITC_AnalogDIntOverUsint
	VAR_INPUT
		IN_Visibility : BOOL;
		IN_ReadOnly : BOOL;
		IN_Wait : BOOL;
		IN_IOType : BOOL; (*0: INPUT 1: OUTPUT*)
		IN_Description : STRING[100];
		IN_MinValue : REAL;
		IN_MaxValue : REAL;
		IN_Unit : STRING[10];
		IN_HMIAutoForce : BOOL;
	END_VAR
	VAR_OUTPUT
		OUT_Man : BOOL;
		OUT_ManValue : DINT;
	END_VAR
	VAR_IN_OUT
		ITC_IO : USINT;
		ITC : DINT;
		HMI_Data : HMI_ITC_Data_Type;
		HMI_Page : HMI_ITC_Page_Type;
		Index : UINT;
	END_VAR
	VAR
		VAR_Man : BOOL := FALSE;
		VAR_RawValue : DINT;
		VAR_Value : DINT;
		VAR_ManValue : DINT := 0;
		VAR_PageSwitch : BOOL := TRUE;
		VAR_ProgressiveId : UINT;
		VAR_OldPage : USINT;
	END_VAR
END_FUNCTION_BLOCK

FUNCTION_BLOCK FB_HMI_ITC_AnalogReal
	VAR_INPUT
		IN_Visibility : BOOL;
		IN_ReadOnly : BOOL;
		IN_Wait : BOOL;
		IN_IOType : BOOL; (*0: INPUT 1: OUTPUT*)
		IN_MinValue : REAL;
		IN_MaxValue : REAL;
		IN_Unit : STRING[10];
		IN_Description : STRING[100];
		IN_HMIAutoForce : BOOL;
	END_VAR
	VAR_OUTPUT
		OUT_Man : BOOL;
		OUT_ManValue : REAL;
	END_VAR
	VAR_IN_OUT
		ITC_IO : REAL;
		ITC : REAL;
		HMI_Data : HMI_ITC_Data_Type;
		HMI_Page : HMI_ITC_Page_Type;
		Index : UINT;
	END_VAR
	VAR
		VAR_Man : BOOL := FALSE;
		VAR_Value : REAL;
		VAR_ManValue : REAL := 0.0;
		VAR_PageSwitch : BOOL := TRUE;
		VAR_ProgressiveId : UINT;
		VAR_OldPage : USINT;
	END_VAR
END_FUNCTION_BLOCK

FUNCTION_BLOCK FB_HMI_ITC_AnalogRealOverUsint
	VAR_INPUT
		IN_Visibility : BOOL;
		IN_ReadOnly : BOOL;
		IN_Wait : BOOL;
		IN_IOType : BOOL; (*0: INPUT 1: OUTPUT*)
		IN_MinValue : REAL;
		IN_MaxValue : REAL;
		IN_Unit : STRING[10];
		IN_Description : STRING[100];
		IN_HMIAutoForce : BOOL;
	END_VAR
	VAR_OUTPUT
		OUT_Man : BOOL;
		OUT_ManValue : REAL;
	END_VAR
	VAR_IN_OUT
		ITC_IO : USINT;
		ITC : REAL;
		HMI_Data : HMI_ITC_Data_Type;
		HMI_Page : HMI_ITC_Page_Type;
		Index : UINT;
	END_VAR
	VAR
		VAR_Man : BOOL := FALSE;
		VAR_RawValue : REAL;
		VAR_Value : REAL;
		VAR_ManValue : REAL := 0.0;
		VAR_PageSwitch : BOOL := TRUE;
		VAR_ProgressiveId : UINT;
		VAR_OldPage : USINT;
		RealValue : REAL;
	END_VAR
END_FUNCTION_BLOCK

FUNCTION_BLOCK FB_HMI_ITC_End
	VAR_INPUT
		IN_IODigAnalog : BOOL; (*0: DIGITAL 1: ANALOG*)
		IN_IOType : BOOL; (*0: INPUT 1: OUTPUT*)
	END_VAR
	VAR_IN_OUT
		HMI_Data : HMI_ITC_Data_Type;
		HMI_Page : HMI_ITC_Page_Type;
		Index : UINT;
	END_VAR
	VAR
		VAR_ProgressiveId : UINT;
		i : UINT;
	END_VAR
END_FUNCTION_BLOCK

FUNCTION_BLOCK FB_HMI_ITC_FastDigitalByte
	VAR_INPUT
		IN_Visibility : BOOL;
		IN_ReadOnly : BOOL;
		IN_Wait : BOOL;
		IN_Alarm : BOOL;
		IN_IOType : BOOL; (*0: INPUT 1: OUTPUT*)
		IN_Description : STRING[100];
		IN_HMIAutoForce : BOOL;
		ITC : BOOL;
	END_VAR
	VAR_OUTPUT
		OUT_Man : BOOL;
		OUT_ManValue : BOOL;
	END_VAR
	VAR_IN_OUT
		HMI_Data : HMI_ITC_Data_Type;
		HMI_Page : HMI_ITC_Page_Type;
		Index : UINT;
	END_VAR
	VAR
		VAR_Auto : BOOL := TRUE;
		VAR_Man : BOOL := FALSE;
		VAR_PageSwitch : BOOL := TRUE;
		VAR_ProgressiveId : UINT;
		VAR_OldPage : USINT;
		zzEdge00000 : BOOL;
		zzEdge00001 : BOOL;
		zzEdge00002 : BOOL;
		zzEdge00003 : BOOL;
	END_VAR
END_FUNCTION_BLOCK

FUNCTION_BLOCK FB_HMI_ITC_FastAnalogInt
	VAR_INPUT
		IN_Visibility : BOOL;
		IN_ReadOnly : BOOL;
		IN_Wait : BOOL;
		IN_IOType : BOOL; (*0: INPUT 1: OUTPUT*)
		IN_Description : STRING[100];
		IN_MinValue : REAL;
		IN_MaxValue : REAL;
		IN_Unit : STRING[10];
		IN_HMIAutoForce : BOOL;
		ITC : INT;
	END_VAR
	VAR_OUTPUT
		OUT_Man : BOOL;
		OUT_ManValue : INT;
	END_VAR
	VAR_IN_OUT
		HMI_Data : HMI_ITC_Data_Type;
		HMI_Page : HMI_ITC_Page_Type;
		Index : UINT;
	END_VAR
	VAR
		VAR_Man : BOOL := FALSE;
		VAR_ManValue : INT := 0;
		VAR_PageSwitch : BOOL := TRUE;
		VAR_ProgressiveId : UINT;
		VAR_OldPage : USINT;
	END_VAR
END_FUNCTION_BLOCK

FUNCTION_BLOCK FB_HMI_ITC_FastAnalogDInt
	VAR_INPUT
		IN_Visibility : BOOL;
		IN_ReadOnly : BOOL;
		IN_Wait : BOOL;
		IN_IOType : BOOL; (*0: INPUT 1: OUTPUT*)
		IN_Description : STRING[100];
		IN_MinValue : REAL;
		IN_MaxValue : REAL;
		IN_Unit : STRING[10];
		IN_HMIAutoForce : BOOL;
		ITC : DINT;
	END_VAR
	VAR_OUTPUT
		OUT_Man : BOOL;
		OUT_ManValue : DINT;
	END_VAR
	VAR_IN_OUT
		HMI_Data : HMI_ITC_Data_Type;
		HMI_Page : HMI_ITC_Page_Type;
		Index : UINT;
	END_VAR
	VAR
		VAR_Man : BOOL := FALSE;
		VAR_ManValue : DINT := 0;
		VAR_PageSwitch : BOOL := TRUE;
		VAR_ProgressiveId : UINT;
		VAR_OldPage : USINT;
	END_VAR
END_FUNCTION_BLOCK

FUNCTION_BLOCK FB_Counter
	VAR_INPUT
		IN_Clock1Hz : BOOL;
		IN_TimeCondition : BOOL;
		IN_IncrementCondition : BOOL;
		IN_PulseWeight : REAL;
		IN_Reset : BOOL;
		IN_Date : DATE_AND_TIME;
	END_VAR
	VAR_IN_OUT
		IN_OUT_CounterPartialStruct : Counters_Type;
		IN_OUT_CounterTotalStruct : Counters_Type;
	END_VAR
	VAR
		tempReal : REAL := 0.0;
	END_VAR
END_FUNCTION_BLOCK

FUNCTION FC_Counter : BOOL (* *) (*$GROUP=User,$CAT=User,$GROUPICON=User.png,$CATICON=User.png*)
	VAR_INPUT
		IN_Clock1Hz : BOOL;
		IN_TimeCondition : BOOL;
		IN_IncrementCondition : BOOL;
		IN_Reset : BOOL;
		IN_Date : DATE_AND_TIME;
	END_VAR
	VAR_IN_OUT
		IN_OUT_CounterPartialStruct : Counters_Type;
		IN_OUT_CounterTotalStruct : Counters_Type;
	END_VAR
END_FUNCTION

FUNCTION FC_IncTimer : BOOL (* *) (*$GROUP=User,$CAT=User,$GROUPICON=User.png,$CATICON=User.png*)
	VAR_INPUT
		IN_Clock1Hz : BOOL;
		IN_Condition : BOOL;
		IN_Reset : BOOL;
	END_VAR
	VAR_IN_OUT
		IN_OUT_CounterStruct : CounterTime_Type;
	END_VAR
END_FUNCTION

FUNCTION FC_SpeedCheck : BOOL (* *) (*$GROUP=User,$CAT=User,$GROUPICON=User.png,$CATICON=User.png*)
	VAR_INPUT
		IN_SpeedReq : REAL;
		IN_SpeedAct : REAL;
		IN_Mode : USINT; (*0 = Equal
1 = Greater
2 = Lower*)
	END_VAR
END_FUNCTION

FUNCTION FC_ReminderShift : INT (*Reminder With Minimum Value*) (*$GROUP=User,$CAT=User,$GROUPICON=User.png,$CATICON=User.png*)
	VAR_INPUT
		Dividend : INT;
		Divisor : INT;
		Start : INT;
	END_VAR
	VAR
		ReminderA : INT;
		ReminderB : INT;
		ReminderC : INT;
		LocalDivisor : INT;
	END_VAR
END_FUNCTION

FUNCTION FC_MacaoTimer : BOOL (* *) (*$GROUP=User,$CAT=User,$GROUPICON=User.png,$CATICON=User.png*)
	VAR_INPUT
		IN_Clock1Hz : BOOL;
		IN_Condition : BOOL;
		IN_Reset : BOOL;
	END_VAR
	VAR_IN_OUT
		IN_OUT_Counter : UDINT;
	END_VAR
END_FUNCTION

FUNCTION_BLOCK Integral
	VAR_INPUT
		IN_NewValue : REAL; (*New value*)
		IN_IntCycle : REAL; (*Cycle time*)
	END_VAR
	VAR_IN_OUT
		OUT_Integral : REAL; (*Integrated value*)
	END_VAR
	VAR
		VAR_OldValue : REAL := 0.0; (*Old value*)
	END_VAR
END_FUNCTION_BLOCK

FUNCTION_BLOCK LevelVariation
	VAR_INPUT
		IN_Enable : BOOL; (*Function Enable*)
		IN_TankVolumePV : REAL; (*Actual Tank Volume [l]*)
		IN_ControlTime : REAL; (*Level Control Scan Time  [s]*)
	END_VAR
	VAR_OUTPUT
		OUT_Low : BOOL; (*Low Flow Required*)
		OUT_High : BOOL; (*High Flow Required*)
	END_VAR
	VAR
		OldVolume : REAL;
		VAR_RTInfo : RTInfo;
		Timer : REAL;
		VAR_Cycle : REAL;
		DeltaVolume : REAL;
		AbsoluteError : REAL; (*Level Error (no sign)*)
		RestoreTime : REAL; (*Number of Cycles with no Negative Variation*)
	END_VAR
	VAR CONSTANT
		RestoreTimeLimit : REAL := 50.0; (*Number of Cycles Limit with no Negative Variation*)
	END_VAR
	VAR
		RestoreError : REAL; (*Number of Cycles in Idle*)
	END_VAR
	VAR CONSTANT
		RestoreErrorLimit : REAL := 50.0; (*Number of Cycles Limit in Idle*)
	END_VAR
END_FUNCTION_BLOCK

FUNCTION_BLOCK PID_Cont
	VAR_INPUT
		IN_ConfigPresent : BOOL; (*Enables PID execution and visualization on HMI*)
		IN_ConfigEngValue : BOOL; (*Configuration: FF and PID OUT Scale - TRUE-> 0-100%, FALSE-> Ing.Unit.*)
		IN_Reverse : BOOL; (*Reverse action (bigger the error smaller the output)*)
		IN_Gain : REAL; (*Proportional gain*)
		IN_TI : REAL; (*Reset time*)
		IN_TD : REAL; (*Derivative time*)
		IN_PV : REAL; (*Process Value for PID Control*)
		IN_Auto : BOOL; (*Execute PID calculations*)
		IN_FixOut : BOOL;
		IN_FixOutValue : REAL;
		IN_IntHold : BOOL; (*Integral action hold*)
		IN_AutoSP : REAL; (*Set Point for PID Control*)
		IN_Disv : REAL; (*Disturbance variable (same unit as manipulated value)*)
		IN_MaxScale : REAL; (*Maximum scale value*)
		IN_Slew : BOOL; (*Slew on SP required*)
		IN_SPSlew : REAL; (*Set Point slew*)
		IN_MinDev : REAL; (*To Set Point Low Deviation (for SP obtained)*)
		IN_MaxDev : REAL; (*To Set Point High Deviation (for SP obtained)*)
		IN_OutMin : REAL; (*Output minimum value*)
		IN_OutMax : REAL; (*Output maximum value*)
		IN_CycleTime : TIME;
		IN_TIInit : BOOL;
		IN_TIInitValue : REAL;
	END_VAR
	VAR_OUTPUT
		OUT : REAL; (*Manipulated value*)
		OUT_ActSP : REAL;
		OUT_Error : REAL; (*Error signal [eng]*)
		OUT_P : REAL; (*Proportionality component*)
		OUT_I : REAL; (*Integral component*)
		OUT_D : REAL; (*Derivative component*)
	END_VAR
	VAR_IN_OUT
		HMI : HMI_PID_Type;
	END_VAR
	VAR
		LCRLimScal_PV : LCRLimScal;
		LCRLimScal_SP : LCRLimScal;
		VAR_Derivative : REAL;
		VAR_FirstCycle : BOOL;
		VAR_GainError : REAL;
		VAR_Integral : Integral;
		VAR_IntegralBlock : BOOL; (*Freeze Integral Calculation*)
		VAR_IntegralOut : REAL;
		VAR_IntegralSaturation : BOOL;
		LCRRamp : LCRRamp;
		VAR_OldError : REAL;
		VAR_Proportional : REAL;
		VAR_RTInfo : RTInfo;
		VAR_SPRamped : REAL;
		VAR_SP : REAL;
		VAR_PV : REAL;
		VAR_CycleCounter : REAL;
		VAR_CycleTime : REAL;
		VAR_SlewInit : BOOL;
		TON_Cycle : TON;
		zzEdge00000 : BOOL;
		zzEdge00001 : BOOL;
		zzEdge00002 : BOOL;
	END_VAR
END_FUNCTION_BLOCK

FUNCTION_BLOCK PID_FF_Mod
	VAR_INPUT
		IN_Enable : BOOL; (*Feed Forward Enable (Bit true)*)
		IN_Reset : BOOL; (*Feed Forward Reset (Bit true)*)
		IN_Raise_Step : REAL; (*Raise Ramp Step Start Delay (0 -:- 100)*)
		IN_Raise_Step_Counter : REAL; (*Raise Ramp Step Start Delay Counter*)
		IN_Lower_Step : REAL; (*Lower  Ramp Step Start Delay (0 -:- 100)*)
		IN_Lower_Step_Counter : REAL; (*Lower Ramp Step Start Delay Counter*)
		IN_FF_SP1 : REAL; (*Feed Forward Set Point 1 Value (High Set Point)*)
		IN_FF_SP2 : REAL; (*Feed Forward Set Point 2 Value (High Set Point)*)
		IN_SP1_SP2_Time : REAL; (*Time delay before Lower Ramp to Feed Forward Set Point 2*)
		IN_Ramp_Speed : REAL; (*Feed Forward Ramp Speed (Raise-Lower)*)
		IN_Actual_Speed : REAL; (*Actual Machine Speed (c/h)*)
		IN_Size_Speed : REAL; (*Max Machine Speed for actual Container Size (c/h)*)
	END_VAR
	VAR_OUTPUT
		OUT_FF_Value : REAL;
		OUT_FF_Value_Int : INT;
	END_VAR
	VAR
		Running : BOOL;
		Lower_Ramp : BOOL;
		SP1_ON : BOOL;
		SP2_ON : BOOL;
		FF_SP1_Recipe : REAL;
		Speed : REAL;
		Max_Speed : REAL;
		FF_SP1_Val : REAL;
		Ramp_Time : REAL;
		Ramp_Speed_R : REAL;
		Ramp_Value : REAL;
		FF_value_Out : REAL;
		FF_SP2_Save : REAL;
		FF_SP2_Time : TON;
		FF_SP2_Recipe : REAL;
		FF_SP2_Val : REAL;
	END_VAR
END_FUNCTION_BLOCK

FUNCTION_BLOCK PID_FF_Pump
	VAR_INPUT
		IN_Enable : BOOL; (*Feed Forward Enable (Bit true)*)
		IN_Reset : BOOL;
		IN_Control_Type : BOOL; (*0=Control on Ring;1=Control on Product Pipe*)
		IN_FV_Number : REAL; (*Filling Valves Number*)
		IN_RingDiameter_mm : REAL;
		IN_FV_FromFloor : REAL; (*Water From The Floor on The Product Level Tank [mm]*)
		IN_PTF_FromFloor : REAL; (*Water From The Floor on The Product Level Tank [mm]*)
		IN_PTF_FromFV : REAL; (*Water From The Floor on The Product Level Tank [mm]*)
		IN_Pump_Kf : REAL;
		IN_Pump_Kpc : REAL;
		IN_Pump_OutMax : REAL;
		IN_FMCActualFlowrate : REAL;
		IN_TankLevel_mm : REAL; (*Water From The Floor on The Product Level Tank [mm]*)
		IN_Actual_SPmm : REAL; (*Actual Machine Speed (B/h)*)
		IN_Actual_PVmm : REAL; (*Actual Machine Speed (B/h)*)
		IN_Actual_SPbar : REAL; (*Actual Machine Speed (B/h)*)
		IN_Actual_PVbar : REAL; (*Actual Machine Speed (B/h)*)
		IN_Actual_Speed : REAL; (*Actual Machine Speed (B/h)*)
	END_VAR
	VAR_OUTPUT
		OUT_FF : REAL;
		OUT_PID_PV : REAL;
		OUT_PID_SP : REAL;
		OUT_Error : BOOL;
	END_VAR
	VAR
		Radius : REAL;
		Omega : REAL;
		CentrifugalForce : REAL;
		Level_SP_Calculated : REAL;
		Pid_PV_Calculated : REAL;
		PV_Product_Pump : REAL;
		Kpc_FlowRate_Filling : REAL;
		Real_Level : REAL;
	END_VAR
END_FUNCTION_BLOCK

FUNCTION_BLOCK PID_FF_PumpH
	VAR_INPUT
		IN_Enable : BOOL; (*Feed Forward Enable (Bit true)*)
		IN_Reset : BOOL;
		IN_Control_Type : BOOL; (*0=Control on Ring;1=Control on Product Pipe*)
		IN_FV_Number : REAL; (*Filling Valves Number*)
		IN_RingDiameter_mm : REAL;
		IN_FV_FromFloor : REAL; (*Water From The Floor on The Product Level Tank [mm]*)
		IN_PTF_FromFloor : REAL; (*Water From The Floor on The Product Level Tank [mm]*)
		IN_PTF_FromFV : REAL; (*Water From The Floor on The Product Level Tank [mm]*)
		IN_Pump_Kf : REAL;
		IN_Pump_Kpc : REAL;
		IN_Pump_OutMax : REAL;
		IN_PumpMaxFillingTime : REAL;
		IN_FMCActualFlowrate : REAL;
		IN_FMCAverFillingTime : REAL;
		IN_FMCStepStartFilling : REAL;
		IN_FMCStepExitCam : REAL;
		IN_TankLevel_mm : REAL; (*Water From The Floor on The Product Level Tank [mm]*)
		IN_Actual_SPmm : REAL; (*Actual Machine Speed (c/h)*)
		IN_Actual_PVmm : REAL; (*Actual Machine Speed (c/h)*)
		IN_Actual_SPbar : REAL; (*Actual Machine Speed (c/h)*)
		IN_Actual_PVbar : REAL; (*Actual Machine Speed (c/h)*)
		IN_Actual_Speed : REAL; (*Actual Machine Speed (c/h)*)
		IN_Recipe_Speed : REAL; (*Max Machine Speed for actual Container Size (c/h)*)
	END_VAR
	VAR_OUTPUT
		OUT_FF : REAL;
		OUT_Centifrugal : REAL;
		OUT_Error : BOOL;
	END_VAR
	VAR
		Radius : REAL;
		Omega : REAL;
		CentrifugalForce : REAL;
		MAX_FillingTime : REAL;
		MAX_ContainersNumber : REAL;
		Level_SP_Calculated : REAL;
		FillingTime : REAL;
		Calculated_FillingTime : REAL;
		PV_Product_Pump : REAL;
		Kpc_FlowRate_Filling : REAL;
		Real_Level : REAL;
	END_VAR
END_FUNCTION_BLOCK

FUNCTION_BLOCK RCP_Management
	VAR_INPUT
		IN_AdrPLCRecipe : {REDUND_UNREPLICABLE} UDINT; (*Temporary structure from HMI*)
		IN_AdrHMIRecipe : {REDUND_UNREPLICABLE} UDINT; (*PLC Internal Structure*)
		IN_SizePLCRecipe : UDINT;
		IN_SizeHMIRecipe : UDINT;
		IN_RequestedRCP : STRING[150];
		IN_DownloadRequest : BOOL;
	END_VAR
	VAR_OUTPUT
		OUT_ParameterError : BOOL;
		OUT_RecipeLoaded : BOOL;
		OUT_Step : RCP_Management_Step;
	END_VAR
	VAR_IN_OUT
		RCP_Manag : RCP_Management_Type;
	END_VAR
	VAR
		VAR_FirstCycle : BOOL;
		VAR_Step_old : RCP_Management_Step;
		TMR_tonRCP_WaitRestart : TON;
		TMR_tonRCP_WaitStart : TON;
		TMR_tonRCP_DownloadTimeOut : TON;
	END_VAR
END_FUNCTION_BLOCK

FUNCTION_BLOCK Sequencer_v1
	VAR_INPUT
		IN_StepConfig : SEQ_StepConfig_Type;
		IN_T_TimeClock : BOOL;
		IN_Step : UINT;
		IN_StepCounter : UINT;
		IN_Pause_Request : BOOL;
		IN_FillingValveNr : UINT;
	END_VAR
	VAR_OUTPUT
		OUT_TON_Time_END : BOOL;
		OUT_TO_Time_END : BOOL;
		OUT_T_Time_END : BOOL;
		OUT_LapsCounterRequest : BOOL;
		OUT_Laps_Done : BOOL;
		OUT_Cycles_Done : BOOL;
		OUT_HMI_ID : UINT; (*ID to match text on HMI*)
		OUT_JMP_StepPrevious : UINT; (*Step wich the sequence is coming from*)
		OUT_JMP_Step : UINT;
		OUT_Laps_Progress : UINT; (*Progress of Laps Executed*)
		OUT_StepTimePr_TON : UINT; (*TON Preset Time*)
		OUT_StepTimePr_T : UINT; (*T Preset Time*)
		OUT_StepTimeCV_TON : UINT; (*TON ActualTime*)
		OUT_StepTimeCV_T : UINT; (*T Actual Time*)
	END_VAR
	VAR_IN_OUT
		CyclesCounter : UDINT;
	END_VAR
	VAR
		TON_Time : TON;
		TO_Time : TON;
		T_Time : CTU;
		VAR_ChangeInProgress : BOOL;
		VAR_CounterInitialized : BOOL;
	END_VAR
END_FUNCTION_BLOCK

FUNCTION_BLOCK Sequencer_v2
	VAR_INPUT
		IN_StepConfig : SEQ_StepConfig_Type;
		IN_T_TimeClock : BOOL;
		IN_Step : UINT;
		IN_StepCounter : UINT;
		IN_Pause_Request : BOOL;
		IN_FillingValveNr : UINT;
	END_VAR
	VAR_OUTPUT
		OUT_TON_Time_END : BOOL;
		OUT_TO_Time_END : BOOL;
		OUT_T_Time_END : BOOL;
		OUT_LapsCounterRequest : BOOL;
		OUT_Laps_Done : BOOL;
		OUT_Cycles_Done : BOOL;
		OUT_HMI_ID : UINT; (*ID to match text on HMI*)
		OUT_StepPrevious : UINT; (*Step wich the sequence is coming from*)
		OUT_StepActual : UINT;
		OUT_Laps_Progress : UINT; (*Progress of Laps Executed*)
		OUT_StepTimePr_TON : UINT; (*TON Preset Time*)
		OUT_StepTimePr_T : UINT; (*T Preset Time*)
		OUT_StepTimeCV_TON : UINT; (*TON ActualTime*)
		OUT_StepTimeCV_T : UINT; (*T Actual Time*)
		OUT_StepProgressiveTime : UINT; (*T Actual Time*)
	END_VAR
	VAR_IN_OUT
		CyclesCounter : UDINT;
	END_VAR
	VAR
		TON_Time : TON;
		TO_Time : TON;
		T_StepProgressiveTime : TON;
		T_Time : CTU;
		VAR_ChangeInProgress : BOOL;
		VAR_CounterInitialized : BOOL;
	END_VAR
END_FUNCTION_BLOCK

FUNCTION_BLOCK TankMultiScale
	VAR_INPUT
		IN_ConfigPresent : BOOL;
		IN_Wait : BOOL;
		IN_Sp_Type : USINT; (*[1=Wait percentage SP] [2=Wait Volume SP] [3=Wait level Height]*)
		IN_TNK_PV : REAL;
		IN_TNK_LowLimitAbs : REAL;
		IN_TNK_Diameter_mm : REAL;
		IN_TNK_Bottom_liters : REAL;
		IN_ProbeLength_mm : REAL;
		IN_FromFloor_ToZeroProbe_mm : REAL;
		IN_Scale : ARRAY[0..3] OF IN_Analog_Multiscale; (*0..3 = Arrays for Different Scale*)
	END_VAR
	VAR_OUTPUT
		OUT_Scale : ARRAY[0..3] OF OUT_Analog_Multiscale;
	END_VAR
	VAR_IN_OUT
		HMI : HMI_Analog_Multiscale_Type;
	END_VAR
	VAR
		pi : REAL;
		diameter_cm : REAL;
		r_cm : REAL; (*radius [cm]*)
		heightAck_cm : REAL;
		volumeAck_cm3 : REAL;
		volumeAck_liters : REAL;
		heightTot_cm : REAL;
		volumeTot_cm3 : REAL;
		volumeTot_liters : REAL;
		LowLimitAbs_cm : REAL;
		LowLimitAbs_cm3 : REAL;
		LowLimitAbs_liters : REAL;
	END_VAR
END_FUNCTION_BLOCK

FUNCTION_BLOCK Siko_Management
	VAR_INPUT
		IN_Mode : INT; (*0: Idle ; 1: Production ; 2: Cleaning*)
		IN_HMI_MotEnable : BOOL;
		IN_HMI_ManualEnable : BOOL;
		IN_HMI_StartWrite : BOOL;
		IN_HMI_Calibrate : BOOL;
		IN_HMI_StartRead : BOOL;
		IN_HMI_JogForward : BOOL;
		IN_HMI_JogBackward : BOOL;
		IN_HMI_MoveAt : BOOL;
		IN_PosProduction : REAL;
		IN_PosCleaning : REAL;
		IN_PosManualSP : REAL;
		IN_EnableToRun : BOOL; (*//v049*)
		IN_Reset : BOOL;
	END_VAR
	VAR_OUTPUT
		OUT_Running : BOOL;
		OUT_Done : BOOL;
		OUT_PositionError : BOOL;
	END_VAR
	VAR_IN_OUT
		IN_SikoData : SIKO_MASTER_Type;
	END_VAR
	VAR
		CalculateSP : REAL;
		Status : INT;
		StepTimer : TON;
		zzEdge00000 : BOOL;
		zzEdge00001 : BOOL;
	END_VAR
END_FUNCTION_BLOCK

FUNCTION_BLOCK Siko_FB
	VAR_INPUT
		IN_EmergencyOK : BOOL;
		IN_Reset : BOOL;
		IN_CommunicationOK : BOOL;
		IN_TimeOutPositioning : TIME;
		IN_PGain : REAL;
		IN_IGain : REAL;
		IN_DGain : REAL;
		IN_VPos : REAL;
		IN_APos : REAL;
		IN_VJog : REAL;
		IN_PosWindows : REAL;
		IN_GearIn : REAL;
		IN_GearOut : REAL;
		IN_SpindlePitch : REAL;
		IN_SenseOfRotation : REAL;
		IN_UpperLimit : REAL;
		IN_LowerLimit : REAL;
		IN_CalibrationValue : REAL;
	END_VAR
	VAR_IN_OUT
		DeviceData : SIKO_MASTER_Type;
		IO : SIKO_COM_Type;
	END_VAR
	VAR
		Com : SIKO_COM_Type;
		ReloadData : BOOL;
		KFactorReal : REAL;
		CounterRead : SINT;
		CounterWrite : SINT;
		CounterCalibration : SINT;
		ReadOrWriteInProgress : BOOL;
		TReadAndWrite : TON;
		zzEdge00000 : BOOL;
		SwitchOn : BOOL;
		TPowerOn : TOF;
		PositionFinished : BOOL;
		zzEdge00001 : BOOL;
		RisingFrontRead : BOOL;
		zzEdge00002 : BOOL;
		RisingFrontWrite : BOOL;
		zzEdge00003 : BOOL;
		zzEdge00004 : BOOL;
		Temp_HIW : UDINT;
		Temp_HSW : UDINT;
		Temp_IN_PWE : UDINT;
		Temp_OUT_PWE : UDINT;
	END_VAR
END_FUNCTION_BLOCK

FUNCTION_BLOCK TP_Reset
	VAR_INPUT
		IN : BOOL;
		PT : TIME;
		RESET : BOOL;
	END_VAR
	VAR_OUTPUT
		Q : BOOL;
	END_VAR
	VAR
		TimeCounter : UDINT;
		RT_Info : RTInfo;
		zzEdge00000 : BOOL;
		zzEdge00001 : BOOL;
	END_VAR
END_FUNCTION_BLOCK

FUNCTION_BLOCK FB_Flip
	VAR_INPUT
		IN_CycleOn : BOOL;
		IN_CyclePause : BOOL;
		IN_CycleLoop : BOOL;
		IN_CycleStartOffCount : BOOL;
		IN_CycleNrReset : BOOL;
		IN_CycleNr : UDINT;
		IN_CycleTimeOn : UDINT;
		IN_CycleTimeOff : UDINT;
	END_VAR
	VAR_OUTPUT
		OUT_CycleNr : UDINT;
		OUT_CycleTimeOn : UDINT;
		OUT_CycleTimeOff : UDINT;
		OUT_CycleDone : BOOL;
		Out : BOOL;
	END_VAR
	VAR
		Command_State : USINT;
		VAR_CycleTimeOn : UDINT;
		VAR_CycleTimeOff : UDINT;
		VAR_CycleNr : UDINT;
		VAR_CyleOn : BOOL;
		VAR_CyleCntOn : BOOL;
		VAR_CyleCntOff : BOOL;
		VAR_CyleOnTimeReset : BOOL;
		VAR_CyleOffTimeReset : BOOL;
		VAR_CyleNrReset : BOOL;
		VAR_CycleOffDone : BOOL;
		VAR_CycleOnDone : BOOL;
		VAR_CycleNrDone : BOOL;
		TON_Blink : TON;
		zzEdge00000 : BOOL;
		zzEdge00001 : BOOL;
		zzEdge00002 : BOOL;
	END_VAR
END_FUNCTION_BLOCK

(* ---- SIKO_FB.st ---- *)
(********************************************************************
 * COPYRIGHT - Sidel SpA
 ********************************************************************
 * Library: SIDEL
 * File: SIKO_FB.st
 * Author: 100383
 * Created: November 16, 2015
 ********************************************************************
 * Implementation of library SIDEL_CNTR
 ********************************************************************)

FUNCTION_BLOCK Siko_FB

	memset(ADR(Com),0,SIZEOF(Com));

	DeviceData.EmergencyOkFbk := IN_EmergencyOK;

	IF NOT IN_CommunicationOK THEN
		DeviceData.PositioningInProgress := FALSE;
		DeviceData.InPosition := FALSE;
		CounterRead := 0;
		CounterWrite := 0;
		DeviceData.CalibrationInProgress := FALSE;
		DeviceData.CommunicationFault := TRUE;
		RETURN;
	ELSE
		DeviceData.CommunicationFault := FALSE;
	END_IF

	IF CounterRead <> 0 OR CounterWrite <> 0 OR (DeviceData.CalibrationInProgress AND NOT DeviceData.Calibrate) THEN
		DeviceData.ReadOrWriteInProgress := TRUE;
	ELSE
		DeviceData.ReadOrWriteInProgress := FALSE;
	END_IF

	TReadAndWrite(IN:= DeviceData.ReadOrWriteInProgress, PT:= t#30s);
	DeviceData.ReadOrWriteError := TReadAndWrite.Q;

	IF DeviceData.ReadOrWriteError OR IN_Reset THEN
		CounterRead := 0;
		CounterWrite := 0;
		DeviceData.CalibrationInProgress := FALSE;
	END_IF

	Com.SIKO_FLR	:= IO.SIKO_FLR;
	Temp_HIW		:= IO.SIKO_FLR.HIW_L + (IO.SIKO_FLR.HIW_H * 16#10000);
	Temp_IN_PWE		:= IO.SIKO_FLR.PWE_L + (IO.SIKO_FLR.PWE_H * 16#10000);

	IF DeviceData.Data.SpindlePitch = 0 THEN
		KFactorReal := 1.0;
	ELSE
		KFactorReal := 100.0;
	END_IF

	DeviceData.CurrentPos := UDINT_TO_REAL(Temp_HIW) / KFactorReal;

	DeviceData.TargetOutsideSwLimit := (DeviceData.TargetPos > DeviceData.Data.UpperLimit) OR (DeviceData.TargetPos < DeviceData.Data.LowerLimit);

	IF EDGEPOS(DeviceData.StartPositioning AND IN_EmergencyOK AND NOT DeviceData.MotorDisabled AND NOT DeviceData.TargetOutsideSwLimit) THEN
		DeviceData.PositioningInProgress := TRUE;
	END_IF

	DeviceData.InPosition := ABS(DeviceData.TargetPos - DeviceData.CurrentPos) <= DeviceData.Data.PosWindows;

	SwitchOn := DeviceData.JogBackward OR DeviceData.JogForward OR DeviceData.PositioningInProgress;

	TPowerOn(IN:= SwitchOn, PT:= t#20s);

	Com.FLR_SIKO.STW.0 := IN_EmergencyOK AND TPowerOn.Q AND DeviceData.Enable AND NOT DeviceData.OnError;
	Com.FLR_SIKO.STW.1 := IN_EmergencyOK AND TPowerOn.Q AND DeviceData.Enable AND NOT DeviceData.OnError;

	Com.FLR_SIKO.STW.7 := IN_Reset;

	Com.FLR_SIKO.STW.5 := Com.SIKO_FLR.ZSW.2 AND NOT DeviceData.AbortPositioning;
	Com.FLR_SIKO.STW.4 := Com.SIKO_FLR.ZSW.2 AND NOT DeviceData.AbortPositioning;

	Com.FLR_SIKO.STW.3 := Com.SIKO_FLR.ZSW.4;

	IF DeviceData.Enable THEN
		DeviceData.MotorDisabled := FALSE;
	ELSIF NOT DeviceData.Enable AND NOT Com.SIKO_FLR.ZSW.4 THEN
		DeviceData.MotorDisabled := TRUE;
	END_IF

	DeviceData.OnError := Com.SIKO_FLR.ZSW.3;

	DeviceData.Warning := Com.SIKO_FLR.ZSW.8 AND Com.SIKO_FLR.ZSW.7;

	DeviceData.DeviceOutsideSwLimit := Com.SIKO_FLR.ZSW.14 OR (DeviceData.CurrentPos > DeviceData.Data.UpperLimit) OR (DeviceData.CurrentPos < DeviceData.Data.LowerLimit);

	Com.FLR_SIKO.STW.9 := Com.SIKO_FLR.ZSW.2 AND NOT DeviceData.OnError AND NOT DeviceData.PositioningInProgress AND	(DeviceData.JogForward XOR DeviceData.JogBackward);

	Com.FLR_SIKO.STW.15 := Com.FLR_SIKO.STW.9 AND DeviceData.JogBackward;

	Com.FLR_SIKO.STW.6 := DeviceData.PositioningInProgress AND NOT DeviceData.OnError AND Com.SIKO_FLR.ZSW.15 AND Com.SIKO_FLR.ZSW.13;

	IF Com.FLR_SIKO.STW.6 THEN
		Temp_HSW := REAL_TO_UDINT(DeviceData.TargetPos * KFactorReal);
	END_IF

	PositionFinished := ABS(DeviceData.TargetPos - DeviceData.CurrentPos) <= DeviceData.Data.PosWindows;

	IF DeviceData.TargetOutsideSwLimit OR DeviceData.OnError OR NOT IN_EmergencyOK OR DeviceData.MotorDisabled OR
	(DeviceData.InPosition AND Com.SIKO_FLR.ZSW.13) OR
	(PositionFinished AND Com.SIKO_FLR.ZSW.13) OR
	EDGEPOS(DeviceData.AbortPositioning) THEN
		DeviceData.PositioningInProgress := FALSE;
	END_IF

	RisingFrontRead := EDGEPOS((DeviceData.StartRead AND NOT DeviceData.ReadOrWriteInProgress) OR ReloadData);

	Com.FLR_SIKO.PKE := 0;

	IF NOT DeviceData.ReadOrWriteError THEN
		IF RisingFrontRead THEN
			CounterRead := 1;
			ReloadData := FALSE;
		END_IF

		CASE CounterRead OF
			1:	// Operative Mode
				Com.FLR_SIKO.PKE := 16#13A2;

				IF Com.SIKO_FLR.PKE = 16#13A2 THEN
					DeviceData.Data.OperationMode := UDINT_TO_INT(Temp_IN_PWE);
					CounterRead := CounterRead  + 1;
				END_IF

			2:	// Error Buffer [0]
				Com.FLR_SIKO.IND := 0;
				Com.FLR_SIKO.PKE := 16#63B1;

				IF Com.SIKO_FLR.PKE = 16#43B1 THEN
					IF Com.SIKO_FLR.IND = 0 THEN
						DeviceData.Data.FaultBuffer0 := UDINT_TO_INT(Temp_IN_PWE);
						CounterRead := CounterRead  + 1;
					END_IF
				END_IF

			3:	// Error Buffer [1]
				Com.FLR_SIKO.IND := 1;
				Com.FLR_SIKO.PKE := 16#63B1;

				IF Com.SIKO_FLR.PKE = 16#43B1 THEN
					IF Com.SIKO_FLR.IND = 1 THEN
						DeviceData.Data.FaultBuffer1 := UDINT_TO_INT(Temp_IN_PWE);
						CounterRead := CounterRead  + 1;
					END_IF
				END_IF

			4:	// Error Buffer [2]
				Com.FLR_SIKO.IND := 2;
				Com.FLR_SIKO.PKE := 16#63B1;

				IF Com.SIKO_FLR.PKE = 16#43B1 THEN
					IF Com.SIKO_FLR.IND = 2 THEN
						DeviceData.Data.FaultBuffer2 := UDINT_TO_INT(Temp_IN_PWE);
						CounterRead := CounterRead  + 1;
					END_IF
				END_IF

			5:	// Error Buffer [3]
				Com.FLR_SIKO.IND := 3;
				Com.FLR_SIKO.PKE := 16#63B1;

				IF Com.SIKO_FLR.PKE = 16#43B1 THEN
					IF Com.SIKO_FLR.IND = 3 THEN
						DeviceData.Data.FaultBuffer3 := UDINT_TO_INT(Temp_IN_PWE);
						CounterRead := CounterRead  + 1;
					END_IF
				END_IF

			6:	// Error Buffer [4]
				Com.FLR_SIKO.IND := 4;
				Com.FLR_SIKO.PKE := 16#63B1;

				IF Com.SIKO_FLR.PKE = 16#43B1 THEN
					IF Com.SIKO_FLR.IND = 4 THEN
						DeviceData.Data.FaultBuffer4 := UDINT_TO_INT(Temp_IN_PWE);
						CounterRead := CounterRead  + 1;
					END_IF
				END_IF

			7:	// Error Buffer [5]
				Com.FLR_SIKO.IND := 5;
				Com.FLR_SIKO.PKE := 16#63B1;

				IF Com.SIKO_FLR.PKE = 16#43B1 THEN
					IF Com.SIKO_FLR.IND = 5 THEN
						DeviceData.Data.FaultBuffer5 := UDINT_TO_INT(Temp_IN_PWE);
						CounterRead := CounterRead  + 1;
					END_IF
				END_IF

			8:	// Error Buffer [6]
				Com.FLR_SIKO.IND := 6;
				Com.FLR_SIKO.PKE := 16#63B1;

				IF Com.SIKO_FLR.PKE = 16#43B1 THEN
					IF Com.SIKO_FLR.IND = 6 THEN
						DeviceData.Data.FaultBuffer6 := UDINT_TO_INT(Temp_IN_PWE);
						CounterRead := CounterRead  + 1;
					END_IF
				END_IF

			9:	// Error Buffer [7]
				Com.FLR_SIKO.IND := 7;
				Com.FLR_SIKO.PKE := 16#63B1;

				IF Com.SIKO_FLR.PKE = 16#43B1 THEN
					IF Com.SIKO_FLR.IND = 7 THEN
						DeviceData.Data.FaultBuffer7 := UDINT_TO_INT(Temp_IN_PWE);
						CounterRead := CounterRead  + 1;
					END_IF
				END_IF

			10:	// Error Buffer [8]
				Com.FLR_SIKO.IND := 8;
				Com.FLR_SIKO.PKE := 16#63B1;

				IF Com.SIKO_FLR.PKE = 16#43B1 THEN
					IF Com.SIKO_FLR.IND = 8 THEN
						DeviceData.Data.FaultBuffer8 := UDINT_TO_INT(Temp_IN_PWE);
						CounterRead := CounterRead  + 1;
					END_IF
				END_IF

			11:	// Error Buffer [9]
				Com.FLR_SIKO.IND := 9;
				Com.FLR_SIKO.PKE := 16#63B1;

				IF Com.SIKO_FLR.PKE = 16#43B1 THEN
					IF Com.SIKO_FLR.IND = 9 THEN
						DeviceData.Data.FaultBuffer9 := UDINT_TO_INT(Temp_IN_PWE);
						CounterRead := CounterRead  + 1;
					END_IF
				END_IF

			12:	// P Gain
				Com.FLR_SIKO.PKE := 16#13E8;

				IF Com.SIKO_FLR.PKE = 16#13E8 THEN
					DeviceData.Data.PGain := UDINT_TO_INT(Temp_IN_PWE);
					CounterRead := CounterRead  + 1;
				END_IF

			13:	// I Gain
				Com.FLR_SIKO.PKE := 16#13E9;

				IF Com.SIKO_FLR.PKE = 16#13E9 THEN
					DeviceData.Data.IGain := UDINT_TO_INT(Temp_IN_PWE);
					CounterRead := CounterRead  + 1;
				END_IF

			14:	// D Gain
				Com.FLR_SIKO.PKE := 16#13EA;

				IF Com.SIKO_FLR.PKE = 16#13EA THEN
					DeviceData.Data.DGain := UDINT_TO_INT(Temp_IN_PWE);
					CounterRead := CounterRead  + 1;
				END_IF

			15:	// A Pos
				Com.FLR_SIKO.PKE := 16#13EB;

				IF Com.SIKO_FLR.PKE = 16#13EB THEN
					DeviceData.Data.APos := UDINT_TO_INT(Temp_IN_PWE);
					CounterRead := CounterRead  + 1;
				END_IF

			16:	// V Pos
				Com.FLR_SIKO.PKE := 16#13EC;

				IF Com.SIKO_FLR.PKE = 16#13EC THEN
					DeviceData.Data.VPos := UDINT_TO_INT(Temp_IN_PWE);
					CounterRead := CounterRead  + 1;
				END_IF

			17:	// V Jog
				Com.FLR_SIKO.PKE := 16#13F0;

				IF Com.SIKO_FLR.PKE = 16#13F0 THEN
					DeviceData.Data.VJog := UDINT_TO_INT(Temp_IN_PWE);
					CounterRead := CounterRead  + 1;
				END_IF

			18:	// SpindlePitch
				Com.FLR_SIKO.PKE := 16#13F4;

				IF Com.SIKO_FLR.PKE = 16#13F4 THEN
					DeviceData.Data.SpindlePitch := UDINT_TO_INT(Temp_IN_PWE) / 100;
					CounterRead := CounterRead  + 1;
				END_IF

			19:	// GearIn
				Com.FLR_SIKO.PKE := 16#13F2;

				IF Com.SIKO_FLR.PKE = 16#13F2 THEN
					DeviceData.Data.GearIn := UDINT_TO_INT(Temp_IN_PWE);
					CounterRead := CounterRead  + 1;
				END_IF

			20:	// GearOut
				Com.FLR_SIKO.PKE := 16#13F3;

				IF Com.SIKO_FLR.PKE = 16#13F3 THEN
					DeviceData.Data.GearOut := UDINT_TO_INT(Temp_IN_PWE);
					CounterRead := CounterRead  + 1;
				END_IF

			21:	// Toll Pos
				Com.FLR_SIKO.PKE := 16#13F1;

				IF Com.SIKO_FLR.PKE = 16#13F1 THEN
					DeviceData.Data.PosWindows := UDINT_TO_REAL(Temp_IN_PWE) / KFactorReal;
					CounterRead := CounterRead  + 1;
				END_IF

			22:	// Rotation
				Com.FLR_SIKO.PKE := 16#13F5;

				IF Com.SIKO_FLR.PKE = 16#13F5 THEN
					DeviceData.Data.SenseOfRotation := UDINT_TO_INT(Temp_IN_PWE);
					CounterRead := CounterRead  + 1;
				END_IF

			23:	// Upper limit
				Com.FLR_SIKO.PKE := 16#13F8;

				IF Com.SIKO_FLR.PKE = 16#13F8 OR Com.SIKO_FLR.PKE = 16#23F8 THEN
					DeviceData.Data.UpperLimit := UDINT_TO_REAL(Temp_IN_PWE) / KFactorReal;
					CounterRead := CounterRead  + 1;
				END_IF

			24:	// Lower limit
				Com.FLR_SIKO.PKE := 16#13F9;

				IF Com.SIKO_FLR.PKE = 16#13F9 OR Com.SIKO_FLR.PKE = 16#23F9 THEN
					DeviceData.Data.LowerLimit := UDINT_TO_REAL(Temp_IN_PWE) / KFactorReal;
					CounterRead := CounterRead  + 1;
				END_IF

			25:	// Calibration value
				Com.FLR_SIKO.PKE := 16#13FA;

				IF Com.SIKO_FLR.PKE = 16#13FA OR Com.SIKO_FLR.PKE = 16#23FA THEN
					DeviceData.Data.CalibrationValue := UDINT_TO_REAL(Temp_IN_PWE) / KFactorReal;
					CounterRead := CounterRead  + 1;
				END_IF

			26:	// Status word
				Com.FLR_SIKO.PKE := 16#13FC;

				IF Com.SIKO_FLR.PKE = 16#13FC THEN
					DeviceData.Data.SystemStatusWord := UDINT_TO_INT(Temp_IN_PWE);
					CounterRead := 0;
				END_IF

		END_CASE
	END_IF

	DeviceData.WriteEnabled := (DeviceData.MotorDisabled OR NOT DeviceData.PositioningInProgress) AND NOT DeviceData.ReadOrWriteInProgress AND NOT DeviceData.ReadOrWriteError AND NOT DeviceData.IllegalOperation;

	RisingFrontWrite := EDGEPOS(DeviceData.StartWrite);

	IF RisingFrontWrite AND DeviceData.WriteEnabled AND NOT DeviceData.ReadOrWriteError THEN
		DeviceData.Data.TimeoutPositioning	:= IN_TimeOutPositioning;
		DeviceData.Data.PosWindows			:= IN_PosWindows;
		DeviceData.Data.UpperLimit			:= IN_UpperLimit;
		DeviceData.Data.LowerLimit			:= IN_LowerLimit;
		DeviceData.Data.CalibrationValue	:= IN_CalibrationValue;

		DeviceData.Data.PGain			:= REAL_TO_INT(IN_PGain);
		DeviceData.Data.IGain			:= REAL_TO_INT(IN_IGain);
		DeviceData.Data.DGain			:= REAL_TO_INT(IN_DGain);
		DeviceData.Data.VPos			:= REAL_TO_INT(IN_VPos);
		DeviceData.Data.APos			:= REAL_TO_INT(IN_APos);
		DeviceData.Data.VJog			:= REAL_TO_INT(IN_VJog);
		DeviceData.Data.GearIn			:= REAL_TO_INT(IN_GearIn);
		DeviceData.Data.GearOut			:= REAL_TO_INT(IN_GearOut);
		DeviceData.Data.SpindlePitch	:= REAL_TO_INT(IN_SpindlePitch);
		DeviceData.Data.SenseOfRotation	:= REAL_TO_INT(IN_SenseOfRotation);
	END_IF

	IF NOT DeviceData.ReadOrWriteError THEN
		IF RisingFrontWrite THEN
			CounterWrite := 1;
		END_IF

		CASE CounterWrite OF
			1:	// Op Mode
				Com.FLR_SIKO.PKE := 16#23A2;
				Temp_OUT_PWE := 2;

				IF Com.SIKO_FLR.PKE = 16#13A2 THEN
					CounterWrite := CounterWrite + 1;
				END_IF

			2:	// Proportional Gain
				Com.FLR_SIKO.PKE := 16#23E8;
				Temp_OUT_PWE := DeviceData.Data.PGain;

				IF Com.SIKO_FLR.PKE = 16#13E8 THEN
					CounterWrite := CounterWrite + 1;
				END_IF

			3:	// Integral Gain
				Com.FLR_SIKO.PKE := 16#23E9;
				Temp_OUT_PWE := DeviceData.Data.IGain;

				IF Com.SIKO_FLR.PKE = 16#13E9 THEN
					CounterWrite := CounterWrite + 1;
				END_IF

			4:	// Derivative Gain
				Com.FLR_SIKO.PKE := 16#23EA;
				Temp_OUT_PWE := DeviceData.Data.DGain;

				IF Com.SIKO_FLR.PKE = 16#13EA THEN
					CounterWrite := CounterWrite + 1;
				END_IF

			5:	// Acc Positioning
				Com.FLR_SIKO.PKE := 16#23EB;
				Temp_OUT_PWE := DeviceData.Data.APos;

				IF Com.SIKO_FLR.PKE = 16#13EB THEN
					CounterWrite := CounterWrite + 1;
				END_IF

			6:	// Speed Positioning
				Com.FLR_SIKO.PKE := 16#23EC;
				Temp_OUT_PWE := DeviceData.Data.VPos;

				IF Com.SIKO_FLR.PKE = 16#13EC THEN
					CounterWrite := CounterWrite + 1;
				END_IF

			7:	// Speed Jog
				Com.FLR_SIKO.PKE := 16#23F0;
				Temp_OUT_PWE := DeviceData.Data.VJog;

				IF Com.SIKO_FLR.PKE = 16#13F0 THEN
					CounterWrite := CounterWrite + 1;
				END_IF

			8:	// GearIn
				Com.FLR_SIKO.PKE := 16#23F2;
				Temp_OUT_PWE := DeviceData.Data.GearIn;

				IF Com.SIKO_FLR.PKE = 16#13F2 THEN
					CounterWrite := CounterWrite + 1;
				END_IF

			9:	// GearOut
				Com.FLR_SIKO.PKE := 16#23F3;
				Temp_OUT_PWE := DeviceData.Data.GearOut;

				IF Com.SIKO_FLR.PKE = 16#13F3 THEN
					CounterWrite := CounterWrite + 1;
				END_IF

			10:	// SpinlePitch
				Com.FLR_SIKO.PKE := 16#23F4;
				Temp_OUT_PWE := DeviceData.Data.SpindlePitch * 100 ;

				IF Com.SIKO_FLR.PKE = 16#13F4 THEN
					CounterWrite := CounterWrite + 1;
				END_IF

			11:	// Position Windows
				Com.FLR_SIKO.PKE := 16#23F1;
				Temp_OUT_PWE := REAL_TO_INT(DeviceData.Data.PosWindows * KFactorReal);

				IF Com.SIKO_FLR.PKE = 16#13F1 THEN
					CounterWrite := CounterWrite + 1;
				END_IF

			12:	// Rotatation
				Com.FLR_SIKO.PKE := 16#23F5;
				Temp_OUT_PWE := DeviceData.Data.SenseOfRotation;

				IF Com.SIKO_FLR.PKE = 16#13F5 THEN
					CounterWrite := CounterWrite + 1;
				END_IF

			13:	// Upper Limit
				Com.FLR_SIKO.PKE := 16#33F8;
				Temp_OUT_PWE := REAL_TO_UDINT(DeviceData.Data.UpperLimit * KFactorReal);

				IF Com.SIKO_FLR.PKE = 16#23F8 THEN
					CounterWrite := CounterWrite + 1;
				ELSIF Com.SIKO_FLR.PKE = 16#73F8 THEN
					CounterWrite := CounterWrite + 2;
				END_IF

			14:	// Lower Limit
				Com.FLR_SIKO.PKE := 16#33F9;
				Temp_OUT_PWE := REAL_TO_UDINT(DeviceData.Data.LowerLimit * KFactorReal);

				IF Com.SIKO_FLR.PKE = 16#23F9 THEN
					CounterWrite := 50;
				END_IF

			15:	//Upper Limit error - Write Lower Limit
				Com.FLR_SIKO.PKE := 16#33F9;
				Temp_OUT_PWE := REAL_TO_UDINT(DeviceData.Data.LowerLimit * KFactorReal);

				IF Com.SIKO_FLR.PKE = 16#23F9 THEN
					CounterWrite := CounterWrite + 1;
				END_IF

			16: //Upper Limit error - Reweite Upper limit
				Com.FLR_SIKO.PKE := 16#33F8;
				Temp_OUT_PWE := REAL_TO_UDINT(DeviceData.Data.UpperLimit * KFactorReal);

				IF Com.SIKO_FLR.PKE = 16#23F8 THEN
					CounterWrite	:= 50;
				END_IF

			50: //Reset PWE
				Temp_OUT_PWE	:= 0;
				CounterWrite	:= 0;
				ReloadData := TRUE;
		END_CASE
	END_IF

	IF EDGEPOS(DeviceData.Calibrate AND DeviceData.WriteEnabled) THEN
		CounterCalibration := 1;
	END_IF

	CASE CounterCalibration OF
		1:
			DeviceData.Data.CalibrationValue := IN_CalibrationValue;
			DeviceData.CalibrationDone := FALSE;
			CounterCalibration := CounterCalibration + 1;

		2://Write Calibration Data
			Com.FLR_SIKO.PKE := 16#33FA;
			Temp_OUT_PWE := REAL_TO_UDINT(DeviceData.Data.CalibrationValue * KFactorReal);
			DeviceData.CalibrationInProgress := TRUE;

			IF Com.SIKO_FLR.PKE = 16#23FA THEN
				CounterCalibration := CounterCalibration + 1;
			END_IF

		3://Check Calibration Data
			IF ABS(Temp_IN_PWE - Temp_HIW) < 5 THEN
				DeviceData.CalibrationDone := TRUE;
				DeviceData.CalibrationInProgress := FALSE;
				CounterCalibration := 0;
			END_IF
	END_CASE

	IF ((DeviceData.Calibrate AND NOT DeviceData.CalibrationInProgress) OR RisingFrontWrite) AND NOT DeviceData.WriteEnabled THEN
		DeviceData.IllegalOperation := TRUE;
	ELSIF DeviceData.IllegalOperation AND IN_Reset THEN
		DeviceData.IllegalOperation := FALSE;
	END_IF

	IO.FLR_SIKO := Com.FLR_SIKO;
	IO.FLR_SIKO.PWE_H := UDINT_TO_UINT(SHR(Temp_OUT_PWE, 16));
	IO.FLR_SIKO.PWE_L := UDINT_TO_UINT(Temp_OUT_PWE AND 16#FFFF);
	IO.FLR_SIKO.HSW_H := UDINT_TO_UINT(SHR(Temp_HSW, 16));
	IO.FLR_SIKO.HSW_L := UDINT_TO_UINT(Temp_HSW AND 16#FFFF) ;

END_FUNCTION_BLOCK

(* ---- Siko_Management.st ---- *)
(********************************************************************
 * COPYRIGHT -- Sidel
 ********************************************************************
 * Library: SIDEL
 * File: Siko_Management.st
 * Author: 100383
 * Created: November 23, 2015
 ********************************************************************
 * Implementation of library SIDEL
 ********************************************************************)

FUNCTION_BLOCK Siko_Management

	IF IN_SikoData.AbortPositioning AND NOT IN_SikoData.PositioningInProgress THEN
		IN_SikoData.AbortPositioning := FALSE;
	END_IF

	IN_SikoData.Enable := IN_HMI_MotEnable;

	IN_SikoData.StartWrite	:= IN_HMI_StartWrite;
	IN_SikoData.Calibrate	:= IN_HMI_Calibrate;
	IN_SikoData.StartRead	:= IN_HMI_StartRead;

	StepTimer();

	CASE IN_Mode OF
		0:
			IN_SikoData.TargetPos	:= IN_SikoData.CurrentPos;

		1:
			IN_SikoData.TargetPos	:= IN_PosProduction;

		2:
			IN_SikoData.TargetPos	:= IN_PosCleaning;

		ELSE
			IN_Mode := 0;
			Status	:= 0;

	END_CASE

	CASE Status OF
		0:		//Ready IDLE
			OUT_Running			:= FALSE;
			OUT_Done			:= FALSE;
			OUT_PositionError	:= FALSE;

			IN_SikoData.StartPositioning := FALSE;

			IN_SikoData.JogBackward    := IN_HMI_JogBackward AND NOT IN_HMI_MoveAt AND IN_HMI_ManualEnable;
			IN_SikoData.JogForward     := IN_HMI_JogForward  AND NOT IN_HMI_MoveAt AND IN_HMI_ManualEnable;

			StepTimer.IN := FALSE;
			StepTimer.PT := t#0s;

			IF IN_Mode = 1  AND NOT IN_HMI_ManualEnable THEN
				Status := 100;
			END_IF

			IF IN_Mode = 2 AND NOT IN_HMI_ManualEnable THEN
				Status := 200;
			END_IF

			IF IN_Mode = 0 AND EDGENEG(IN_HMI_MoveAt) AND NOT IN_HMI_JogForward AND NOT IN_HMI_JogBackward AND IN_HMI_ManualEnable THEN
				IN_SikoData.TargetPos := IN_PosManualSP;
				Status	:= 10;
			END_IF

		10:		//Manual positioning
			OUT_Running			:= FALSE;
			OUT_Done			:= FALSE;
			OUT_PositionError	:= FALSE;

			StepTimer.IN	:= TRUE;
			StepTimer.PT	:= t#240s;

			IN_SikoData.StartPositioning	:=	IN_SikoData.CalibrationDone			AND NOT IN_SikoData.OnError					AND NOT
												IN_SikoData.CommunicationFault		AND NOT IN_SikoData.MotorDisabled			AND IN_SikoData.EmergencyOkFbk	AND NOT
												IN_SikoData.TargetOutsideSwLimit	AND NOT IN_SikoData.DeviceOutsideSwLimit;

			IN_SikoData.TargetPos			:= IN_PosManualSP;

			//Motor in position
			IF IN_SikoData.InPosition THEN
				IN_SikoData.StartPositioning := FALSE;
				StepTimer.IN := FALSE;
				Status := 0;
			END_IF

			//Timeout positioning or change modality
			IF StepTimer.Q OR EDGEPOS(IN_HMI_MoveAt) OR NOT IN_HMI_ManualEnable OR IN_Mode <> 0 THEN
				IN_SikoData.StartPositioning := FALSE;
				IN_SikoData.AbortPositioning := TRUE;
				StepTimer.IN := FALSE;
				Status := 20;
			END_IF

		20:		//Abort command. Wait 0.5s motor stop before changing mode or make a new operation
			OUT_Running			:= FALSE;
			OUT_Done			:= FALSE;
			OUT_PositionError	:= FALSE;

			StepTimer.IN	:= TRUE;
			StepTimer.PT	:= t#0.5s;

			IN_SikoData.StartPositioning := FALSE;

			IF StepTimer.Q AND NOT IN_HMI_MoveAt THEN
				IN_SikoData.AbortPositioning := FALSE;
				StepTimer.IN := FALSE;
				Status := 0;
			END_IF

		100:	//Production
			OUT_Running			:= TRUE;
			OUT_Done			:= FALSE;
			OUT_PositionError	:= FALSE;

			OUT_PositionError := FALSE;

			IN_SikoData.StartPositioning := FALSE;

			IF IN_Mode <> 1 THEN
				StepTimer.IN := FALSE;
				Status := 0;
			END_IF

			IF IN_SikoData.MotorDisabled THEN
				StepTimer.IN := FALSE;
				Status := 150;
			END_IF

			IF IN_SikoData.InPosition THEN
				OUT_Done := TRUE;
				StepTimer.IN := FALSE;
				Status := 120;
			ELSE
				IF NOT IN_SikoData.PositioningInProgress AND IN_EnableToRun THEN //v049
					StepTimer.IN := FALSE;
					Status := 110;
				END_IF
			END_IF

		110:	//Production - Wait for positioning
			OUT_Running			:= TRUE;
			OUT_Done			:= FALSE;
			OUT_PositionError	:= FALSE;

			StepTimer.PT	:= t#240s;

			OUT_PositionError := FALSE;

			IN_SikoData.StartPositioning := IN_SikoData.CalibrationDone			AND NOT IN_SikoData.OnError					AND NOT
											IN_SikoData.CommunicationFault		AND NOT IN_SikoData.MotorDisabled			AND IN_SikoData.EmergencyOkFbk	AND NOT
											IN_SikoData.TargetOutsideSwLimit	AND NOT IN_SikoData.DeviceOutsideSwLimit;

			StepTimer.IN := IN_SikoData.StartPositioning;

			//Motor in position
			IF IN_SikoData.InPosition THEN
				StepTimer.IN := FALSE;
				Status := 120;
			END_IF

			IF IN_SikoData.OnError OR StepTimer.Q OR IN_SikoData.CommunicationFault OR IN_SikoData.TargetOutsideSwLimit THEN
				IN_SikoData.AbortPositioning := TRUE;
				IN_SikoData.StartPositioning := FALSE;
				StepTimer.IN := FALSE;
				Status := 130;
			END_IF

			IF NOT IN_SikoData.EmergencyOkFbk THEN
				IN_SikoData.StartPositioning := FALSE;
				StepTimer.IN := FALSE;
				Status := 140;
			END_IF

			IF IN_SikoData.MotorDisabled THEN
				StepTimer.IN := FALSE;
				Status := 150;
			END_IF

			IF IN_Mode <> 1 THEN
				StepTimer.IN := FALSE;
				Status := 190;
			END_IF

		120:	//Motor in position
			OUT_Running			:= TRUE;
			OUT_Done			:= TRUE;
			OUT_PositionError	:= FALSE;

			IN_SikoData.StartPositioning := FALSE;
			StepTimer.IN	:= FALSE;

			IF NOT IN_SikoData.InPosition THEN
				Status := 160;
			END_IF

			IF IN_SikoData.MotorDisabled THEN
				Status := 150;
			END_IF

			IF IN_Mode <> 1 THEN
				Status := 0;
			END_IF

		130:	//Error during positioning phase. Aknoledge required
			OUT_Running			:= TRUE;
			OUT_Done			:= FALSE;
			OUT_PositionError	:= TRUE;

			IN_SikoData.StartPositioning := FALSE;
			StepTimer.IN	:= FALSE;

			IF IN_Reset THEN
				IN_SikoData.AbortPositioning := FALSE;
				OUT_PositionError := FALSE;
				Status := 100;
			END_IF

			IF IN_HMI_MoveAt THEN
				IN_SikoData.AbortPositioning := FALSE;
				OUT_PositionError := FALSE;
				Status := 131;
			END_IF

			IF IN_SikoData.MotorDisabled THEN
				IN_SikoData.AbortPositioning := FALSE;
				OUT_PositionError := FALSE;
				Status := 150;
			END_IF

			IF IN_Mode <> 1 THEN
				IN_SikoData.AbortPositioning :=FALSE;
				StepTimer.PT :=FALSE;
				Status :=0;
			END_IF

		131: 	//Error during positioning phase. Manual positioning
			OUT_Running			:= TRUE;
			OUT_Done			:= FALSE;
			OUT_PositionError	:= FALSE;

			IN_SikoData.StartPositioning := FALSE;
			StepTimer.IN	:= TRUE;
			StepTimer.PT	:= t#240s;

			IN_SikoData.StartPositioning := IN_SikoData.CalibrationDone			AND NOT IN_SikoData.OnError					AND NOT
											IN_SikoData.CommunicationFault		AND NOT IN_SikoData.MotorDisabled			AND IN_SikoData.EmergencyOkFbk	AND NOT
											IN_SikoData.TargetOutsideSwLimit	AND NOT IN_SikoData.DeviceOutsideSwLimit;

			//Motor in position
			IF IN_SikoData.InPosition AND NOT IN_HMI_MoveAt THEN
				IN_SikoData.StartPositioning := FALSE;
				StepTimer.IN := FALSE;
				Status := 120;
			END_IF

			//Timeout positioning
			IF StepTimer.Q THEN
				IN_SikoData.StartPositioning := FALSE;
				IN_SikoData.AbortPositioning := TRUE;
				StepTimer.IN := FALSE;
				Status := 130;
			END_IF

			IF IN_SikoData.MotorDisabled THEN
				IN_SikoData.AbortPositioning := TRUE;
				OUT_PositionError := FALSE;
				Status := 150;
			END_IF

			IF IN_Mode <> 1 THEN
				IN_SikoData.StartPositioning := FALSE;
				IN_SikoData.AbortPositioning := TRUE;
				StepTimer.IN := FALSE;
				Status := 132;
			END_IF

		132:		//Abort command. Wait 0.5s before changing mode or make a new operation
			OUT_Running			:= TRUE;
			OUT_Done			:= FALSE;
			OUT_PositionError	:= FALSE;

			StepTimer.IN	:= TRUE;
			StepTimer.PT	:= t#0.5s;

			IN_SikoData.StartPositioning := FALSE;

			IF StepTimer.Q AND NOT IN_HMI_MoveAt THEN
				IN_SikoData.AbortPositioning := FALSE;
				StepTimer.IN := FALSE;
				Status := 0;
			END_IF

		140:	//Emergency
			OUT_Running			:= TRUE;
			OUT_Done			:= FALSE;
			OUT_PositionError	:= FALSE;

			IN_SikoData.StartPositioning := FALSE;

			IF IN_SikoData.EmergencyOkFbk THEN
				StepTimer.IN := FALSE;
				Status := 100;
			END_IF

			IF IN_SikoData.MotorDisabled THEN
				Status := 150;
			END_IF

			IF IN_Mode <> 1 THEN
				Status := 0;
			END_IF

		150:	//Motor disabled
			OUT_Running			:= TRUE;
			OUT_Done			:= FALSE;
			OUT_PositionError	:= FALSE;

			IN_SikoData.StartPositioning := FALSE;
			IN_SikoData.AbortPositioning := FALSE;

			IF NOT IN_SikoData.MotorDisabled THEN
				StepTimer.IN := FALSE;
				Status := 130;
			END_IF

			IF IN_Mode <> 1 THEN
				Status := 0;
			END_IF

		160:	//Positioning lost
			OUT_Running			:= TRUE;
			OUT_Done			:= FALSE;
			OUT_PositionError	:= FALSE;

			IF IN_SikoData.MotorDisabled OR IN_Reset THEN
				StepTimer.IN := FALSE;
				Status := 100;
			END_IF

			IF IN_Mode <> 1 THEN
				Status := 0;
			END_IF

		190: //Exit step
			OUT_Running			:= FALSE;
			OUT_Done			:= FALSE;
			OUT_PositionError	:= FALSE;

			StepTimer.IN := TRUE;
			StepTimer.PT := t#2s;

			IN_SikoData.AbortPositioning := TRUE;
			IN_SikoData.StartPositioning := FALSE;

			IF StepTimer.Q AND NOT IN_HMI_MoveAt THEN
				IN_SikoData.AbortPositioning := FALSE;
				StepTimer.IN := FALSE;
				Status	:= 0;
			END_IF

		200:	//Cleaning
			OUT_Running			:= TRUE;
			OUT_Done			:= FALSE;
			OUT_PositionError	:= FALSE;

			IN_SikoData.StartPositioning := FALSE;

			IF IN_Mode <> 2 THEN
				StepTimer.IN := FALSE;
				Status := 0;
			END_IF

			IF IN_SikoData.MotorDisabled THEN
				StepTimer.IN := FALSE;
				Status := 250;
			END_IF

			IF IN_SikoData.InPosition THEN
				OUT_Done := TRUE;
				StepTimer.IN := FALSE;
				Status := 220;
			ELSE
				IF NOT IN_SikoData.PositioningInProgress AND IN_EnableToRun THEN //v049
					StepTimer.IN := FALSE;
					Status := 210;
				END_IF
			END_IF

		210:	//Cleaning - Wait for position
			OUT_Running			:= TRUE;
			OUT_Done			:= FALSE;
			OUT_PositionError	:= FALSE;

			StepTimer.PT := t#240s;

			IN_SikoData.StartPositioning := IN_SikoData.CalibrationDone			AND NOT IN_SikoData.OnError					AND NOT
											IN_SikoData.CommunicationFault		AND NOT IN_SikoData.MotorDisabled			AND IN_SikoData.EmergencyOkFbk	AND NOT
											IN_SikoData.TargetOutsideSwLimit	AND NOT IN_SikoData.DeviceOutsideSwLimit;

			StepTimer.IN := IN_SikoData.StartPositioning;

			IF IN_SikoData.InPosition THEN
				StepTimer.IN := FALSE;
				Status := 220;
			END_IF

			IF IN_SikoData.OnError OR StepTimer.Q OR IN_SikoData.CommunicationFault OR IN_SikoData.TargetOutsideSwLimit THEN
				IN_SikoData.AbortPositioning := TRUE;
				IN_SikoData.StartPositioning := FALSE;
				StepTimer.IN := FALSE;
				Status := 230;
			END_IF

			IF NOT IN_SikoData.EmergencyOkFbk THEN
				IN_SikoData.StartPositioning := FALSE;
				StepTimer.IN := FALSE;
				Status := 240;
			END_IF

			IF IN_SikoData.MotorDisabled THEN
				StepTimer.IN := FALSE;
				Status := 250;
			END_IF

			IF IN_Mode <> 2 THEN
				StepTimer.IN := FALSE;
				Status := 290;
			END_IF

		220: 	//Motor in position
			OUT_Running			:= TRUE;
			OUT_Done			:= TRUE;
			OUT_PositionError	:= FALSE;

			IN_SikoData.StartPositioning := FALSE;
			StepTimer.IN := FALSE;

			IF NOT IN_SikoData.InPosition THEN
				Status := 260;
			END_IF

			IF IN_SikoData.MotorDisabled THEN
				Status := 250;
			END_IF

			IF IN_Mode <> 2 THEN
				Status := 0;
			END_IF

		230:
			OUT_Running			:= TRUE;
			OUT_Done			:= FALSE;
			OUT_PositionError	:= TRUE;

			IN_SikoData.StartPositioning := FALSE;
			StepTimer.IN	:= FALSE;

			IF IN_Reset THEN
				IN_SikoData.AbortPositioning := FALSE;
				OUT_PositionError := FALSE;
				Status := 200;
			END_IF

			IF IN_HMI_MoveAt THEN
				IN_SikoData.AbortPositioning := FALSE;
				OUT_PositionError := FALSE;
				Status := 231;
			END_IF

			IF IN_SikoData.MotorDisabled THEN
				IN_SikoData.AbortPositioning := FALSE;
				OUT_PositionError := FALSE;
				Status := 250;
			END_IF

			IF IN_Mode <> 2 THEN
				IN_SikoData.AbortPositioning :=FALSE;
				StepTimer.PT :=FALSE;
				Status :=0;
			END_IF

		231: 	//Error during positioning phase. Manual positioning
			OUT_Running			:= TRUE;
			OUT_Done			:= FALSE;
			OUT_PositionError	:= FALSE;

			IN_SikoData.StartPositioning := FALSE;
			StepTimer.IN	:= TRUE;
			StepTimer.PT	:= t#240s;

			IN_SikoData.StartPositioning := IN_SikoData.CalibrationDone			AND NOT IN_SikoData.OnError					AND NOT
											IN_SikoData.CommunicationFault		AND NOT IN_SikoData.MotorDisabled			AND IN_SikoData.EmergencyOkFbk	AND NOT
											IN_SikoData.TargetOutsideSwLimit	AND NOT IN_SikoData.DeviceOutsideSwLimit;

			//Motor in position
			IF IN_SikoData.InPosition AND NOT IN_HMI_MoveAt THEN
				IN_SikoData.StartPositioning := FALSE;
				StepTimer.IN := FALSE;
				Status := 220;
			END_IF

			//Timeout positioning
			IF StepTimer.Q THEN
				IN_SikoData.StartPositioning := FALSE;
				IN_SikoData.AbortPositioning := TRUE;
				StepTimer.IN := FALSE;
				Status := 230;
			END_IF

			IF IN_SikoData.MotorDisabled THEN
				IN_SikoData.AbortPositioning := TRUE;
				OUT_PositionError := FALSE;
				Status := 250;
			END_IF

			IF IN_Mode <> 1 THEN
				IN_SikoData.StartPositioning := FALSE;
				IN_SikoData.AbortPositioning := TRUE;
				StepTimer.IN := FALSE;
				Status := 232;
			END_IF

		232:		//Abort command. Wait 0.5s before changing mode or make a new operation
			OUT_Running			:= TRUE;
			OUT_Done			:= FALSE;
			OUT_PositionError	:= FALSE;

			StepTimer.IN	:= TRUE;
			StepTimer.PT	:= t#0.5s;

			IN_SikoData.StartPositioning := FALSE;

			IF StepTimer.Q AND NOT IN_HMI_MoveAt THEN
				IN_SikoData.AbortPositioning := FALSE;
				StepTimer.IN := FALSE;
				Status := 0;
			END_IF

		240: 	//Emergency
			OUT_Running			:= TRUE;
			OUT_Done			:= FALSE;
			OUT_PositionError	:= FALSE;

			IN_SikoData.StartPositioning := FALSE;

			IF IN_SikoData.EmergencyOkFbk THEN
				StepTimer.IN := FALSE;
				Status := 200;
			END_IF

			IF IN_SikoData.MotorDisabled THEN
				Status := 250;
			END_IF

			IF IN_Mode <> 2 THEN
				Status := 0;
			END_IF

		250:	//Motor disabled
			OUT_Running			:= TRUE;
			OUT_Done			:= FALSE;
			OUT_PositionError	:= FALSE;

			IN_SikoData.StartPositioning := FALSE;
			IN_SikoData.AbortPositioning := FALSE;

			IF NOT IN_SikoData.MotorDisabled THEN
				StepTimer.IN := FALSE;
				Status := 230;
			END_IF

			IF IN_Mode <> 2 THEN
				Status := 0;
			END_IF

		260:	//Positioning lost
			OUT_Running			:= TRUE;
			OUT_Done			:= FALSE;
			OUT_PositionError	:= FALSE;

			IF IN_SikoData.MotorDisabled OR IN_Reset THEN
				StepTimer.IN := FALSE;
				Status := 200;
			END_IF

			IF IN_Mode <> 2 THEN
				Status := 0;
			END_IF

		290: //Exit step.
			OUT_Running			:= FALSE;
			OUT_Done			:= FALSE;
			OUT_PositionError	:= FALSE;

			StepTimer.IN := TRUE;
			StepTimer.PT := t#2s;

			IN_SikoData.AbortPositioning := TRUE;
			IN_SikoData.StartPositioning := FALSE;

			IF StepTimer.Q AND NOT IN_HMI_MoveAt THEN
				IN_SikoData.AbortPositioning := FALSE;
				StepTimer.IN := FALSE;
				Status	:= 0;
			END_IF

		ELSE
			Status := 0;
	END_CASE
END_FUNCTION_BLOCK

(* ---- TankLevel.st ---- *)
FUNCTION_BLOCK TankMultiScale
	IF IN_ProbeLength_mm = 0.0 OR IN_TNK_Diameter_mm = 0.0 THEN
		RETURN;
	END_IF

	//Index [0]: level in percentage
	//Index [1]: volume in liters
	//Index [2]: height in mm
	//Index [3]: HMI_PAR_2._309

	pi 			:= 3.14;
	diameter_cm	:= IN_TNK_Diameter_mm / 10.0; 	// [cm]
	r_cm  		:= diameter_cm / 2.0;			// [cm]

	heightTot_cm		:= IN_ProbeLength_mm / 10.0; 	// [cm]
	volumeTot_cm3 		:= (pi * r_cm * r_cm) * heightTot_cm;	// [cm3]
	volumeTot_liters 	:= volumeTot_cm3 / 1000;			// [dm3]/[l]

	heightAck_cm		:= IN_ProbeLength_mm / 10.0 * IN_TNK_PV / 100.0;	// [cm]
	volumeAck_cm3 		:= (pi * r_cm * r_cm) * heightAck_cm;	// [cm3]
	volumeAck_liters 	:= volumeAck_cm3 / 1000;			// [dm3]/[l]

	LowLimitAbs_cm		:= IN_ProbeLength_mm / 10.0 * IN_TNK_LowLimitAbs / 100.0;	// [cm]
	LowLimitAbs_cm3		:= (pi * r_cm * r_cm) * LowLimitAbs_cm;	// [cm3]
	LowLimitAbs_liters 	:= LowLimitAbs_cm3 / 1000;			// [dm3]/[l]

	OUT_Scale[0].ActValue	:=	LIMIT(IN_Scale[0].ScaleLOW, IN_TNK_PV, IN_Scale[0].ScaleHIGH);
	IF IN_TNK_PV > 1.0 THEN
		OUT_Scale[1].ActValue := volumeAck_liters + IN_TNK_Bottom_liters;
	ELSE
		OUT_Scale[1].ActValue := 0.0;
	END_IF

	OUT_Scale[2].ActValue 	:= (OUT_Scale[0].ActValue * IN_ProbeLength_mm / 100.0)(* + IN_FromFloor_ToZeroProbe_mm*);

	OUT_Scale[3].ActValue := LowLimitAbs_liters + IN_TNK_Bottom_liters;

	CASE IN_Sp_Type OF
		0:
			HMI.SP[0] 		:= IN_Scale[0].ActualSP;
			HMI.SP[1]		:= IN_Scale[1].ActualSP;
			HMI.SP[2]		:= IN_Scale[2].ActualSP;
			HMI.SP[3]		:= IN_Scale[3].ActualSP;
			HMI.Wait[0] 	:= FALSE;
			HMI.Wait[1]		:= FALSE;
			HMI.Wait[2]		:= FALSE;
			HMI.Wait[3]		:= FALSE;

		1:	// Wait percentage SP
			HMI.SP[0] 		:= IN_Scale[0].ActualSP;
			HMI.SP[1]		:= (IN_Scale[0].ActualSP * volumeTot_liters) / 100.0;
			HMI.SP[2]		:= (IN_Scale[0].ActualSP * IN_ProbeLength_mm / 100.0) + IN_FromFloor_ToZeroProbe_mm;
			HMI.SP[3]		:= IN_Scale[3].ActualSP;
			HMI.Wait[0] 	:= IN_Wait;
			HMI.Wait[1]		:= FALSE;
			HMI.Wait[2]		:= FALSE;
			HMI.Wait[3]		:= FALSE;

		2:	// Wait Volume SP
			HMI.SP[0]		:= ((IN_Scale[1].ActualSP - IN_TNK_Bottom_liters) / volumeTot_liters) *100.0;
			HMI.SP[1]		:= IN_Scale[1].ActualSP;
			HMI.SP[2]		:= (((IN_Scale[1].ActualSP / volumeTot_liters) *100.0) * IN_ProbeLength_mm /100.0) + IN_FromFloor_ToZeroProbe_mm;
			HMI.SP[3]		:= IN_Scale[3].ActualSP;
			HMI.Wait[0] 	:= FALSE;
			HMI.Wait[1]		:= IN_Wait;
			HMI.Wait[2]		:= FALSE;
			HMI.Wait[3]		:= FALSE;

		3:	// Wait level Height
			HMI.SP[0] 		:= (IN_Scale[2].ActualSP - IN_FromFloor_ToZeroProbe_mm) / IN_ProbeLength_mm  *100.0;
			HMI.SP[1]		:= (HMI.SP[0] * volumeTot_liters) / 100.0 + IN_TNK_Bottom_liters;
			HMI.SP[2]		:= IN_Scale[2].ActualSP;
			HMI.SP[3]		:= IN_Scale[3].ActualSP;
			HMI.Wait[0] 	:= FALSE;
			HMI.Wait[1]		:= FALSE;
			HMI.Wait[2]		:= IN_Wait;
			HMI.Wait[3]		:= FALSE;
	END_CASE

	HMI.ConfigPresent	:= IN_ConfigPresent;
	HMI.PV[0] 			:= OUT_Scale[0].ActValue;
	HMI.PV[1] 			:= OUT_Scale[1].ActValue;
	HMI.PV[2] 			:= OUT_Scale[2].ActValue;
	HMI.PV[3] 			:= OUT_Scale[3].ActValue;

END_FUNCTION_BLOCK

(* ---- TP_Reset.st ---- *)
FUNCTION_BLOCK TP_Reset
	RT_Info(enable := TRUE);

	IF EDGEPOS(IN) THEN
		TimeCounter	:= TIME_TO_UDINT(PT) * 1000;	//micros
	END_IF

	IF TimeCounter >= RT_Info.cycle_time THEN
		TimeCounter := TimeCounter - (RT_Info.cycle_time);
	ELSE
		TimeCounter := 0;
	END_IF

	IF EDGEPOS(RESET) THEN
		TimeCounter := 0;
	END_IF

	Q := TimeCounter <> 0;
END_FUNCTION_BLOCK

(* ---- Constant.var ---- *)
(*ITC*)
VAR CONSTANT
	CST_MinITCPartner : USINT := 11;
	CST_MaxITCPartner : USINT := 89; (*V4.A.A.1.6.12*)
END_VAR
(*HMI Rele Station and Channel State*)
VAR CONSTANT
	CST_MAX_Nr_Channels : USINT := 16;
	CST_RELE_NO_COMMUN : USINT := 0; (*White + X Red Symbol*)
	CST_RELE_ON : USINT := 1; (*Green*)
	CST_RELE_ON_BY_PLC : USINT := 2; (*Green*)
	CST_RELE_ON_WARNING : USINT := 3; (*Green + Warning Symbol*)
	CST_RELE_ON_CONFIG_ERROR : USINT := 4; (*Green + Yellow with X Blue*)
	CST_RELE_OFF_FAULT : USINT := 5; (*Black + Fault Symbol*)
	CST_RELE_OFF_BY_PB_HW : USINT := 6; (*Black + HW Symbol*)
	CST_RELE_OFF_BY_HMI : USINT := 7; (*Black + HMI Symbol*)
	CST_RELE_OFF_BY_PLC : USINT := 8; (*Black + PLC Symbol*)
	CST_RELE_OFF : USINT := 9; (*Black*)
	CST_RELE_OFF_CONFIG_ERROR : USINT := 10; (*Black + Yellow with X Blue*)
	CST_RELE_NOT_DEFINE : USINT := 11; (*Yellow + X Blue*)
END_VAR
